# B&R Automation Studio project NAEUL004C00R13L518F00 (part 16)

#### Act_OptP0923Navi.st
```iecst
ACTION Act_OptP0923Navi:

	IF tyP0923SafetyBar.tyNaviBack.tyBtnBack.bRtCompl = TRUE OR tyP0923SafetyBar.tyNaviLyr1.tyBtnBack.bRtCompl = TRUE OR tyP0923SafetyBar.tyNaviLyr2.tyBtnBack.bRtCompl = TRUE THEN
		tyP0923SafetyBar.tyNaviBack.tyBtnBack.bRtCompl 	:= FALSE;
		tyP0923SafetyBar.tyNaviBack.tyBtnBack.bValue	:= FALSE;
		tyP0923SafetyBar.tyNaviLyr1.tyBtnBack.bRtCompl 	:= FALSE;
		tyP0923SafetyBar.tyNaviLyr1.tyBtnBack.bValue	:= FALSE;
		tyP0923SafetyBar.tyNaviLyr2.tyBtnBack.bRtCompl 	:= FALSE;
		tyP0923SafetyBar.tyNaviLyr2.tyBtnBack.bValue	:= FALSE;

		eChgPage	:= UIP0920MtrNPneuCtrl;

	ELSIF tyP0923SafetyBar.tyNaviLyr1.tyBtnLeft.bRtCompl = TRUE OR tyP0923SafetyBar.tyNaviLyr1.tyBtnRgt.bRtCompl = TRUE THEN
		tyP0923SafetyBar.tyNaviLyr1.tyBtnLeft.bRtCompl	:= FALSE;
		tyP0923SafetyBar.tyNaviLyr1.tyBtnRgt.bRtCompl	:= FALSE;

		bDispSafetyBar1	:= FALSE;
		bDispSafetyBar2	:= TRUE;

		p_tyC0004Navi ACCESS ADR(tyP0923SafetyBar.tyNaviLyr2);

		p_tyP0923LftSafetyBarCom ACCESS ADR(tyP0923SafetyBar.tyMag3SafetyBarCom);
		p_tyP0923LftSafetyBarDC ACCESS ADR(tyP0923SafetyBar.tyMag3SafetyBarDC);
		p_tyP0923LftSafetyBarFB ACCESS ADR(tyP0923SafetyBar.tyMag3SafetyBarFB);

		p_tyP0923RgtSafetyBarCom ACCESS ADR(tyP0923SafetyBar.tyRgtSafetyBarComHide);
		p_tyP0923RgtSafetyBarDC ACCESS ADR(tyP0923SafetyBar.tyRgtSafetyBarDCHide);
		p_tyP0923RgtSafetyBarFB ACCESS ADR(tyP0923SafetyBar.tyRgtSafetyBarFBHide);

	ELSIF tyP0923SafetyBar.tyNaviLyr2.tyBtnLeft.bRtCompl = TRUE OR tyP0923SafetyBar.tyNaviLyr2.tyBtnRgt.bRtCompl = TRUE THEN
		tyP0923SafetyBar.tyNaviLyr2.tyBtnLeft.bRtCompl	:= FALSE;
		tyP0923SafetyBar.tyNaviLyr2.tyBtnRgt.bRtCompl	:= FALSE;

		bDispSafetyBar1	:= TRUE;
		bDispSafetyBar2	:= FALSE;

		p_tyC0004Navi ACCESS ADR(tyP0923SafetyBar.tyNaviLyr1);

		p_tyP0923LftSafetyBarCom ACCESS ADR(tyP0923SafetyBar.tyMag1SafetyBarCom);
		p_tyP0923LftSafetyBarDC ACCESS ADR(tyP0923SafetyBar.tyMag1SafetyBarDC);
		p_tyP0923LftSafetyBarFB ACCESS ADR(tyP0923SafetyBar.tyMag1SafetyBarFB);

		p_tyP0923RgtSafetyBarCom ACCESS ADR(tyP0923SafetyBar.tyMag2SafetyBarCom);
		p_tyP0923RgtSafetyBarDC ACCESS ADR(tyP0923SafetyBar.tyMag2SafetyBarDC);
		p_tyP0923RgtSafetyBarFB ACCESS ADR(tyP0923SafetyBar.tyMag2SafetyBarFB);

	END_IF

END_ACTION
```

#### Act_OptP0923DualMask.st
```iecst
ACTION Act_OptP0923DualMask:

	IF eCurrPage = UIP0923SafetyBar THEN

		IF p_tyDI.bEStopSig = FALSE THEN
			p_tyC0003DualMask ACCESS ADR(tyP0923SafetyBar.tyDualMaskEStop);

			tyP0923SafetyBar.tyDualMaskEStop.tyBtnLeftMask.uiMaskRtStat.0	:= FALSE;
			tyP0923SafetyBar.tyDualMaskEStop.tyBtnRgtMask.uiMaskRtStat.0	:= bDispSafetyBar2;

		ELSIF p_tyDI.bCoverSWSig = FALSE THEN
			p_tyC0003DualMask ACCESS ADR(tyP0923SafetyBar.tyDualMaskCWSig);

			tyP0923SafetyBar.tyDualMaskCWSig.tyBtnLeftMask.uiMaskRtStat.0	:= FALSE;
			tyP0923SafetyBar.tyDualMaskCWSig.tyBtnRgtMask.uiMaskRtStat.0	:= bDispSafetyBar2;

		ELSIF p_tyDI.bSafetyRlySig = FALSE THEN
			p_tyC0003DualMask ACCESS ADR(tyP0923SafetyBar.tyDualMaskSafetyRly);

			tyP0923SafetyBar.tyDualMaskSafetyRly.tyBtnLeftMask.uiMaskRtStat.0	:= FALSE;
			tyP0923SafetyBar.tyDualMaskSafetyRly.tyBtnRgtMask.uiMaskRtStat.0	:= bDispSafetyBar2;

//		ELSIF p_tyDI.bPusherRetRS = FALSE THEN
//			p_tyC0003DualMask ACCESS ADR(tyP0923SafetyBar.tyDualMaskPshrInterrupt);
//
//			tyP0923SafetyBar.tyDualMaskPshrInterrupt.tyBtnLeftMask.uiMaskRtStat.0	:= FALSE;
//			tyP0923SafetyBar.tyDualMaskPshrInterrupt.tyBtnRgtMask.uiMaskRtStat.0	:= bDispSafetyBar2;
//
		ELSE
			p_tyC0003DualMask ACCESS ADR(tyP0923SafetyBar.tyDualMaskHide);

		END_IF

	END_IF

END_ACTION
```

#### Act_OptP0923Mag1SafetyBarChgLyr.st
```iecst
ACTION Act_OptP0923Mag1SafetyBarChgLyr:

	IF tyP0923SafetyBar.tyMag1SafetyBarCom.tyBtnSwitch.bRtCompl THEN
		tyP0923SafetyBar.tyMag1SafetyBarCom.tyBtnSwitch.bRtCompl := FALSE;

		IF tyP0923SafetyBar.tyMag1SafetyBarCom.tyBtnSwitch.bValue = TRUE THEN
			fUIInRtStatOff(ADR(tyP0923SafetyBar.tyMag1SafetyBarDC.tyLyr.uiRtStat));
			fUIInRtStatHide(ADR(tyP0923SafetyBar.tyMag1SafetyBarFB.tyLyr.uiRtStat));
		ELSE
			fUIInRtStatHide(ADR(tyP0923SafetyBar.tyMag1SafetyBarDC.tyLyr.uiRtStat));
			fUIInRtStatOff(ADR(tyP0923SafetyBar.tyMag1SafetyBarFB.tyLyr.uiRtStat));
		END_IF

	END_IF

END_ACTION
```

#### Act_OptP0923Mag1SafetyBarSen.st
```iecst
ACTION Act_OptP0923Mag1SafetyBarSen:

	tyP0923SafetyBar.tyMag1SafetyBarCom.tyBtnExtRS.bValue	:= p_tyDI.bMag1SafetyBarExtRS;
	tyP0923SafetyBar.tyMag1SafetyBarCom.tyBtnRetRS.bValue	:= p_tyDI.bMag1SafetyBarRetRS;

	//Machine Bitmap
	IF p_tyDI.bMag1SafetyBarRetRS = TRUE THEN
		tyP0923SafetyBar.tyMag1SafetyBarCom.tyBitmapMc.uiValueIdx	:= 1;
	ELSE
		tyP0923SafetyBar.tyMag1SafetyBarCom.tyBitmapMc.uiValueIdx	:= 0;
	END_IF

	IF p_tyNtParamCurr.eProjMag = ULMagTriple THEN
		IF p_tyNtParamCurr.bProjMagAWPrep = FALSE AND p_tyNtParamCurr.bProjMotorizedPusherPrep = FALSE THEN
		IF 	tyP0923SafetyBar.tyMag1SafetyBarCom.tyBitmapMc.uiValueIdx < 100 THEN
			tyP0923SafetyBar.tyMag1SafetyBarCom.tyBitmapMc.uiValueIdx	:= tyP0923SafetyBar.tyMag1SafetyBarCom.tyBitmapMc.uiValueIdx + 100;
		END_IF
	ELSIF p_tyNtParamCurr.bProjMagAWPrep = FALSE AND p_tyNtParamCurr.bProjMotorizedPusherPrep = TRUE THEN
		IF 	tyP0923SafetyBar.tyMag1SafetyBarCom.tyBitmapMc.uiValueIdx < 400 THEN
		tyP0923SafetyBar.tyMag1SafetyBarCom.tyBitmapMc.uiValueIdx	:= tyP0923SafetyBar.tyMag1SafetyBarCom.tyBitmapMc.uiValueIdx + 400;
		END_IF
		END_IF
		END_IF
END_ACTION
```

#### Act_OptP0923Mag1SafetyBarFB.st
```iecst
ACTION Act_OptP0923Mag1SafetyBarFB:

	IF tyP0923SafetyBar.tyMag1SafetyBarCom.tyBtnSwitch.bValue = FALSE THEN

		IF tyP0923SafetyBar.tyMag1SafetyBarFB.tyBtnRet.bRtCompl = TRUE THEN
			tyP0923SafetyBar.tyMag1SafetyBarFB.tyBtnRet.bRtCompl	:= FALSE;

			tyP0923SafetyBar.tyMag1SafetyBarFB.tyBtnRet.bValue		:= TRUE;
			tyP0923SafetyBar.tyMag1SafetyBarFB.tyBtnExt.bValue		:= FALSE;

		ELSIF tyP0923SafetyBar.tyMag1SafetyBarFB.tyBtnExt.bRtCompl = TRUE THEN
			tyP0923SafetyBar.tyMag1SafetyBarFB.tyBtnExt.bRtCompl	:= FALSE;

			tyP0923SafetyBar.tyMag1SafetyBarFB.tyBtnExt.bValue		:= TRUE;
			tyP0923SafetyBar.tyMag1SafetyBarFB.tyBtnRet.bValue		:= FALSE;
		END_IF

		IF tyP0923SafetyBar.tyMag1SafetyBarFB.tyBtnRet.bValue = TRUE THEN
			eMag1SafetyBarAct	:= PneuActRet;

			IF p_eMag1SafetyBarStat = PneuActRet AND p_eMag1SafetyBarStatus = Done THEN
				eMag1SafetyBarAct	:= PneuActIdle;

				tyP0923SafetyBar.tyMag1SafetyBarFB.tyBtnRet.bValue	:= FALSE;
			ELSIF p_eMag1SafetyBarStatus = Error THEN
				tyP0923SafetyBar.tyMag1SafetyBarFB.tyBtnRet.bValue	:= FALSE;
			END_IF

		ELSIF tyP0923SafetyBar.tyMag1SafetyBarFB.tyBtnExt.bValue = TRUE THEN
			eMag1SafetyBarAct	:= PneuActExt;

			IF p_eMag1SafetyBarStat = PneuActExt AND p_eMag1SafetyBarStatus = Done THEN
				eMag1SafetyBarAct	:= PneuActIdle;

				tyP0923SafetyBar.tyMag1SafetyBarFB.tyBtnExt.bValue := FALSE;
			ELSIF p_eMag1SafetyBarStatus = Error THEN
				tyP0923SafetyBar.tyMag1SafetyBarFB.tyBtnExt.bValue := FALSE;
			END_IF
		END_IF

		//Update Direct Control Status
		tyP0923SafetyBar.tyMag1SafetyBarDC.tyBtnRet.bRtCompl	:= FALSE;
		tyP0923SafetyBar.tyMag1SafetyBarDC.tyBtnExt.bRtCompl	:= FALSE;
		tyP0923SafetyBar.tyMag1SafetyBarDC.tyBtnRet.bValue		:= p_bMag1SafetyBarRetCtrl;
		tyP0923SafetyBar.tyMag1SafetyBarDC.tyBtnExt.bValue		:= p_bMag1SafetyBarExtCtrl;

	END_IF

END_ACTION
```

#### Act_OptP0923Mag1SafetyBarFBStat.st
```iecst
ACTION Act_OptP0923Mag1SafetyBarFBStat:

	tyP0923SafetyBar.tyMag1SafetyBarFB.tyStringStat.sValue	:= p_sMag1SafetyBarStatTxt;

END_ACTION
```

#### Act_OptP0923Mag1SafetyBarDC.st
```iecst
ACTION Act_OptP0923Mag1SafetyBarDC:

	IF tyP0923SafetyBar.tyMag1SafetyBarCom.tyBtnSwitch.bValue = TRUE THEN

		IF p_bMag1SafetyBarTwoCtrlOut = FALSE THEN

			IF tyP0923SafetyBar.tyMag1SafetyBarDC.tyBtnRet.bRtCompl = TRUE THEN
				tyP0923SafetyBar.tyMag1SafetyBarDC.tyBtnRet.bValue	:= TRUE;
				tyP0923SafetyBar.tyMag1SafetyBarDC.tyBtnExt.bValue	:= FALSE;

				eMag1SafetyBarAct	:= PneuActSetRet;

				IF p_eMag1SafetyBarStat = PneuActSetRet AND p_eMag1SafetyBarStatus = Done THEN
					eMag1SafetyBarAct	:= PneuActIdle;

					tyP0923SafetyBar.tyMag1SafetyBarDC.tyBtnRet.bRtCompl	:= FALSE;
				END_IF

			ELSIF tyP0923SafetyBar.tyMag1SafetyBarDC.tyBtnExt.bRtCompl = TRUE THEN
				tyP0923SafetyBar.tyMag1SafetyBarDC.tyBtnExt.bValue	:= TRUE;
				tyP0923SafetyBar.tyMag1SafetyBarDC.tyBtnRet.bValue	:= FALSE;

				eMag1SafetyBarAct	:= PneuActSetExt;

				IF p_eMag1SafetyBarStat = PneuActSetExt AND p_eMag1SafetyBarStatus = Done THEN
					eMag1SafetyBarAct	:= PneuActIdle;

					tyP0923SafetyBar.tyMag1SafetyBarDC.tyBtnExt.bRtCompl	:= FALSE;
				END_IF

			END_IF

		ELSE

			IF (tyP0923SafetyBar.tyMag1SafetyBarDC.tyBtnRet.bRtCompl = TRUE) OR (tyP0923SafetyBar.tyMag1SafetyBarDC.tyBtnExt.bRtCompl = TRUE) THEN

				IF (tyP0923SafetyBar.tyMag1SafetyBarDC.tyBtnRet.bValue = TRUE) AND (tyP0923SafetyBar.tyMag1SafetyBarDC.tyBtnExt.bValue = TRUE) THEN
					eMag1SafetyBarAct	:= PneuActSetAll;

					IF p_eMag1SafetyBarStat = PneuActSetAll AND p_eMag1SafetyBarStatus = Done THEN
						eMag1SafetyBarAct	:= PneuActIdle;

						tyP0923SafetyBar.tyMag1SafetyBarDC.tyBtnRet.bRtCompl	:= FALSE;
						tyP0923SafetyBar.tyMag1SafetyBarDC.tyBtnExt.bRtCompl	:= FALSE;
					END_IF

				ELSIF (tyP0923SafetyBar.tyMag1SafetyBarDC.tyBtnRet.bValue = TRUE) AND (tyP0923SafetyBar.tyMag1SafetyBarDC.tyBtnExt.bValue = FALSE) THEN
					eMag1SafetyBarAct	:= PneuActSetRet;

					IF p_eMag1SafetyBarStat = PneuActSetRet AND p_eMag1SafetyBarStatus = Done THEN
						eMag1SafetyBarAct	:= PneuActIdle;

						tyP0923SafetyBar.tyMag1SafetyBarDC.tyBtnRet.bRtCompl	:= FALSE;
						tyP0923SafetyBar.tyMag1SafetyBarDC.tyBtnExt.bRtCompl	:= FALSE;
					END_IF

				ELSIF (tyP0923SafetyBar.tyMag1SafetyBarDC.tyBtnRet.bValue = FALSE) AND (tyP0923SafetyBar.tyMag1SafetyBarDC.tyBtnExt.bValue = TRUE) THEN
					eMag1SafetyBarAct	:= PneuActSetExt;

					IF p_eMag1SafetyBarStat = PneuActSetExt AND p_eMag1SafetyBarStatus = Done THEN
						eMag1SafetyBarAct	:= PneuActIdle;

						tyP0923SafetyBar.tyMag1SafetyBarDC.tyBtnRet.bRtCompl	:= FALSE;
						tyP0923SafetyBar.tyMag1SafetyBarDC.tyBtnExt.bRtCompl	:= FALSE;
					END_IF

				ELSE
					eMag1SafetyBarAct	:= PneuActRstAll;

					IF p_eMag1SafetyBarStat = PneuActRstAll AND p_eMag1SafetyBarStatus = Done THEN
						eMag1SafetyBarAct	:= PneuActIdle;

						tyP0923SafetyBar.tyMag1SafetyBarDC.tyBtnRet.bRtCompl	:= FALSE;
						tyP0923SafetyBar.tyMag1SafetyBarDC.tyBtnExt.bRtCompl	:= FALSE;
					END_IF

				END_IF

			END_IF

		END_IF

		tyP0923SafetyBar.tyMag1SafetyBarFB.tyBtnExt.bRtCompl	:= FALSE;
		tyP0923SafetyBar.tyMag1SafetyBarFB.tyBtnExt.bValue		:= FALSE;
		tyP0923SafetyBar.tyMag1SafetyBarFB.tyBtnRet.bRtCompl	:= FALSE;
		tyP0923SafetyBar.tyMag1SafetyBarFB.tyBtnRet.bValue		:= FALSE;

	END_IF

END_ACTION
```

#### Act_OptP0923Mag2SafetyBarChgLyr.st
```iecst
ACTION Act_OptP0923Mag2SafetyBarChgLyr:

	IF tyP0923SafetyBar.tyMag2SafetyBarCom.tyBtnSwitch.bRtCompl THEN
		tyP0923SafetyBar.tyMag2SafetyBarCom.tyBtnSwitch.bRtCompl := FALSE;

		IF tyP0923SafetyBar.tyMag2SafetyBarCom.tyBtnSwitch.bValue = TRUE THEN
			fUIInRtStatOff(ADR(tyP0923SafetyBar.tyMag2SafetyBarDC.tyLyr.uiRtStat));
			fUIInRtStatHide(ADR(tyP0923SafetyBar.tyMag2SafetyBarFB.tyLyr.uiRtStat));
		ELSE
			fUIInRtStatHide(ADR(tyP0923SafetyBar.tyMag2SafetyBarDC.tyLyr.uiRtStat));
			fUIInRtStatOff(ADR(tyP0923SafetyBar.tyMag2SafetyBarFB.tyLyr.uiRtStat));
		END_IF

	END_IF

END_ACTION
```

#### Act_OptP0923Mag2SafetyBarSen.st
```iecst
ACTION Act_OptP0923Mag2SafetyBarSen:

	tyP0923SafetyBar.tyMag2SafetyBarCom.tyBtnExtRS.bValue	:= p_tyDI.bMag2SafetyBarExtRS;
	tyP0923SafetyBar.tyMag2SafetyBarCom.tyBtnRetRS.bValue	:= p_tyDI.bMag2SafetyBarRetRS;

	//Machine Bitmap
	IF p_tyDI.bMag2SafetyBarRetRS = TRUE THEN
		tyP0923SafetyBar.tyMag2SafetyBarCom.tyBitmapMc.uiValueIdx	:= 3;
	ELSE
		tyP0923SafetyBar.tyMag2SafetyBarCom.tyBitmapMc.uiValueIdx	:= 2;
	END_IF

	IF p_tyNtParamCurr.eProjMag = ULMagTriple THEN
		IF p_tyNtParamCurr.bProjMagAWPrep = FALSE AND p_tyNtParamCurr.bProjMotorizedPusherPrep = FALSE THEN
		IF 	tyP0923SafetyBar.tyMag2SafetyBarCom.tyBitmapMc.uiValueIdx < 100 THEN
				tyP0923SafetyBar.tyMag2SafetyBarCom.tyBitmapMc.usiValueIdx	:= tyP0923SafetyBar.tyMag2SafetyBarCom.tyBitmapMc.usiValueIdx + 100;
				END_IF
	ELSIF p_tyNtParamCurr.bProjMagAWPrep = FALSE AND p_tyNtParamCurr.bProjMotorizedPusherPrep = TRUE THEN
		IF 	tyP0923SafetyBar.tyMag2SafetyBarCom.tyBitmapMc.uiValueIdx < 400 THEN
			tyP0923SafetyBar.tyMag2SafetyBarCom.tyBitmapMc.uiValueIdx	:= tyP0923SafetyBar.tyMag2SafetyBarCom.tyBitmapMc.uiValueIdx + 400;
		END_IF
			END_IF
			END_IF
END_ACTION
```

#### Act_OptP0923Mag2SafetyBarFB.st
```iecst
ACTION Act_OptP0923Mag2SafetyBarFB:

	IF tyP0923SafetyBar.tyMag2SafetyBarCom.tyBtnSwitch.bValue = FALSE THEN

		IF tyP0923SafetyBar.tyMag2SafetyBarFB.tyBtnRet.bRtCompl = TRUE THEN
			tyP0923SafetyBar.tyMag2SafetyBarFB.tyBtnRet.bRtCompl	:= FALSE;

			tyP0923SafetyBar.tyMag2SafetyBarFB.tyBtnRet.bValue		:= TRUE;
			tyP0923SafetyBar.tyMag2SafetyBarFB.tyBtnExt.bValue		:= FALSE;

		ELSIF tyP0923SafetyBar.tyMag2SafetyBarFB.tyBtnExt.bRtCompl = TRUE THEN
			tyP0923SafetyBar.tyMag2SafetyBarFB.tyBtnExt.bRtCompl	:= FALSE;

			tyP0923SafetyBar.tyMag2SafetyBarFB.tyBtnExt.bValue		:= TRUE;
			tyP0923SafetyBar.tyMag2SafetyBarFB.tyBtnRet.bValue		:= FALSE;
		END_IF

		IF tyP0923SafetyBar.tyMag2SafetyBarFB.tyBtnRet.bValue = TRUE THEN
			eMag2SafetyBarAct	:= PneuActRet;

			IF p_eMag2SafetyBarStat = PneuActRet AND p_eMag2SafetyBarStatus = Done THEN
				eMag2SafetyBarAct	:= PneuActIdle;

				tyP0923SafetyBar.tyMag2SafetyBarFB.tyBtnRet.bValue	:= FALSE;
			ELSIF p_eMag2SafetyBarStatus = Error THEN
				tyP0923SafetyBar.tyMag2SafetyBarFB.tyBtnRet.bValue	:= FALSE;
			END_IF

		ELSIF tyP0923SafetyBar.tyMag2SafetyBarFB.tyBtnExt.bValue = TRUE THEN
			eMag2SafetyBarAct	:= PneuActExt;

			IF p_eMag2SafetyBarStat = PneuActExt AND p_eMag2SafetyBarStatus = Done THEN
				eMag2SafetyBarAct	:= PneuActIdle;

				tyP0923SafetyBar.tyMag2SafetyBarFB.tyBtnExt.bValue := FALSE;
			ELSIF p_eMag2SafetyBarStatus = Error THEN
				tyP0923SafetyBar.tyMag2SafetyBarFB.tyBtnExt.bValue := FALSE;
			END_IF
		END_IF

		//Update Direct Control Status
		tyP0923SafetyBar.tyMag2SafetyBarDC.tyBtnRet.bRtCompl	:= FALSE;
		tyP0923SafetyBar.tyMag2SafetyBarDC.tyBtnExt.bRtCompl	:= FALSE;
		tyP0923SafetyBar.tyMag2SafetyBarDC.tyBtnRet.bValue		:= p_bMag2SafetyBarRetCtrl;
		tyP0923SafetyBar.tyMag2SafetyBarDC.tyBtnExt.bValue		:= p_bMag2SafetyBarExtCtrl;

	END_IF

END_ACTION
```

#### Act_OptP0923Mag2SafetyBarFBStat.st
```iecst
ACTION Act_OptP0923Mag2SafetyBarFBStat:

	tyP0923SafetyBar.tyMag2SafetyBarFB.tyStringStat.sValue	:= p_sMag2SafetyBarStatTxt;

END_ACTION
```

#### Act_OptP0923Mag2SafetyBarDC.st
```iecst
ACTION Act_OptP0923Mag2SafetyBarDC:

	IF tyP0923SafetyBar.tyMag2SafetyBarCom.tyBtnSwitch.bValue = TRUE THEN

		IF p_bMag2SafetyBarTwoCtrlOut = FALSE THEN

			IF tyP0923SafetyBar.tyMag2SafetyBarDC.tyBtnRet.bRtCompl = TRUE THEN
				tyP0923SafetyBar.tyMag2SafetyBarDC.tyBtnRet.bValue	:= TRUE;
				tyP0923SafetyBar.tyMag2SafetyBarDC.tyBtnExt.bValue	:= FALSE;

				eMag2SafetyBarAct	:= PneuActSetRet;

				IF p_eMag2SafetyBarStat = PneuActSetRet AND p_eMag2SafetyBarStatus = Done THEN
					eMag2SafetyBarAct	:= PneuActIdle;

					tyP0923SafetyBar.tyMag2SafetyBarDC.tyBtnRet.bRtCompl	:= FALSE;
				END_IF

			ELSIF tyP0923SafetyBar.tyMag2SafetyBarDC.tyBtnExt.bRtCompl = TRUE THEN
				tyP0923SafetyBar.tyMag2SafetyBarDC.tyBtnExt.bValue	:= TRUE;
				tyP0923SafetyBar.tyMag2SafetyBarDC.tyBtnRet.bValue	:= FALSE;

				eMag2SafetyBarAct	:= PneuActSetExt;

				IF p_eMag2SafetyBarStat = PneuActSetExt AND p_eMag2SafetyBarStatus = Done THEN
					eMag2SafetyBarAct	:= PneuActIdle;

					tyP0923SafetyBar.tyMag2SafetyBarDC.tyBtnExt.bRtCompl	:= FALSE;
				END_IF

			END_IF

		ELSE

			IF (tyP0923SafetyBar.tyMag2SafetyBarDC.tyBtnRet.bRtCompl = TRUE) OR (tyP0923SafetyBar.tyMag2SafetyBarDC.tyBtnExt.bRtCompl = TRUE) THEN

				IF (tyP0923SafetyBar.tyMag2SafetyBarDC.tyBtnRet.bValue = TRUE) AND (tyP0923SafetyBar.tyMag2SafetyBarDC.tyBtnExt.bValue = TRUE) THEN
					eMag2SafetyBarAct	:= PneuActSetAll;

					IF p_eMag2SafetyBarStat = PneuActSetAll AND p_eMag2SafetyBarStatus = Done THEN
						eMag2SafetyBarAct	:= PneuActIdle;

						tyP0923SafetyBar.tyMag2SafetyBarDC.tyBtnRet.bRtCompl	:= FALSE;
						tyP0923SafetyBar.tyMag2SafetyBarDC.tyBtnExt.bRtCompl	:= FALSE;
					END_IF

				ELSIF (tyP0923SafetyBar.tyMag2SafetyBarDC.tyBtnRet.bValue = TRUE) AND (tyP0923SafetyBar.tyMag2SafetyBarDC.tyBtnExt.bValue = FALSE) THEN
					eMag2SafetyBarAct	:= PneuActSetRet;

					IF p_eMag2SafetyBarStat = PneuActSetRet AND p_eMag2SafetyBarStatus = Done THEN
						eMag2SafetyBarAct	:= PneuActIdle;

						tyP0923SafetyBar.tyMag2SafetyBarDC.tyBtnRet.bRtCompl	:= FALSE;
						tyP0923SafetyBar.tyMag2SafetyBarDC.tyBtnExt.bRtCompl	:= FALSE;
					END_IF

				ELSIF (tyP0923SafetyBar.tyMag2SafetyBarDC.tyBtnRet.bValue = FALSE) AND (tyP0923SafetyBar.tyMag2SafetyBarDC.tyBtnExt.bValue = TRUE) THEN
					eMag2SafetyBarAct	:= PneuActSetExt;

					IF p_eMag2SafetyBarStat = PneuActSetExt AND p_eMag2SafetyBarStatus = Done THEN
						eMag2SafetyBarAct	:= PneuActIdle;

						tyP0923SafetyBar.tyMag2SafetyBarDC.tyBtnRet.bRtCompl	:= FALSE;
						tyP0923SafetyBar.tyMag2SafetyBarDC.tyBtnExt.bRtCompl	:= FALSE;
					END_IF

				ELSE
					eMag2SafetyBarAct	:= PneuActRstAll;

					IF p_eMag2SafetyBarStat = PneuActRstAll AND p_eMag2SafetyBarStatus = Done THEN
						eMag2SafetyBarAct	:= PneuActIdle;

						tyP0923SafetyBar.tyMag2SafetyBarDC.tyBtnRet.bRtCompl	:= FALSE;
						tyP0923SafetyBar.tyMag2SafetyBarDC.tyBtnExt.bRtCompl	:= FALSE;
					END_IF

				END_IF

			END_IF

		END_IF

		tyP0923SafetyBar.tyMag2SafetyBarFB.tyBtnExt.bRtCompl	:= FALSE;
		tyP0923SafetyBar.tyMag2SafetyBarFB.tyBtnExt.bValue		:= FALSE;
		tyP0923SafetyBar.tyMag2SafetyBarFB.tyBtnRet.bRtCompl	:= FALSE;
		tyP0923SafetyBar.tyMag2SafetyBarFB.tyBtnRet.bValue		:= FALSE;

	END_IF

END_ACTION
```

#### Act_OptP0923Mag3SafetyBarChgLyr.st
```iecst
ACTION Act_OptP0923Mag3SafetyBarChgLyr:

	IF tyP0923SafetyBar.tyMag3SafetyBarCom.tyBtnSwitch.bRtCompl THEN
		tyP0923SafetyBar.tyMag3SafetyBarCom.tyBtnSwitch.bRtCompl := FALSE;

		IF tyP0923SafetyBar.tyMag3SafetyBarCom.tyBtnSwitch.bValue = TRUE THEN
			fUIInRtStatOff(ADR(tyP0923SafetyBar.tyMag3SafetyBarDC.tyLyr.uiRtStat));
			fUIInRtStatHide(ADR(tyP0923SafetyBar.tyMag3SafetyBarFB.tyLyr.uiRtStat));
		ELSE
			fUIInRtStatHide(ADR(tyP0923SafetyBar.tyMag3SafetyBarDC.tyLyr.uiRtStat));
			fUIInRtStatOff(ADR(tyP0923SafetyBar.tyMag3SafetyBarFB.tyLyr.uiRtStat));
		END_IF

	END_IF

END_ACTION
```

#### Act_OptP0923Mag3SafetyBarSen.st
```iecst
ACTION Act_OptP0923Mag3SafetyBarSen:

	tyP0923SafetyBar.tyMag3SafetyBarCom.tyBtnExtRS.bValue	:= p_tyDI.bMag3SafetyBarExtRS;
	tyP0923SafetyBar.tyMag3SafetyBarCom.tyBtnRetRS.bValue	:= p_tyDI.bMag3SafetyBarRetRS;

	//Machine Bitmap
	IF p_tyDI.bMag3SafetyBarRetRS = TRUE THEN
		tyP0923SafetyBar.tyMag3SafetyBarCom.tyBitmapMc.uiValueIdx	:= 5;
	ELSE
		tyP0923SafetyBar.tyMag3SafetyBarCom.tyBitmapMc.uiValueIdx	:= 4;
	END_IF

	IF p_tyNtParamCurr.eProjMag = ULMagTriple THEN
		IF p_tyNtParamCurr.bProjMagAWPrep = FALSE AND p_tyNtParamCurr.bProjMotorizedPusherPrep = FALSE THEN
		IF 	tyP0923SafetyBar.tyMag3SafetyBarCom.tyBitmapMc.uiValueIdx < 100 THEN
		tyP0923SafetyBar.tyMag3SafetyBarCom.tyBitmapMc.usiValueIdx	:= tyP0923SafetyBar.tyMag3SafetyBarCom.tyBitmapMc.usiValueIdx + 100;
		END_IF
		ELSIF p_tyNtParamCurr.bProjMagAWPrep = FALSE AND p_tyNtParamCurr.bProjMotorizedPusherPrep = TRUE THEN
		IF 	tyP0923SafetyBar.tyMag3SafetyBarCom.tyBitmapMc.uiValueIdx < 400 THEN
			tyP0923SafetyBar.tyMag3SafetyBarCom.tyBitmapMc.uiValueIdx	:= tyP0923SafetyBar.tyMag3SafetyBarCom.tyBitmapMc.uiValueIdx + 400;
		END_IF
		END_IF
		END_IF
END_ACTION
```

#### Act_OptP0923Mag3SafetyBarFB.st
```iecst
ACTION Act_OptP0923Mag3SafetyBarFB:

	IF tyP0923SafetyBar.tyMag3SafetyBarCom.tyBtnSwitch.bValue = FALSE THEN

		IF tyP0923SafetyBar.tyMag3SafetyBarFB.tyBtnRet.bRtCompl = TRUE THEN
			tyP0923SafetyBar.tyMag3SafetyBarFB.tyBtnRet.bRtCompl	:= FALSE;

			tyP0923SafetyBar.tyMag3SafetyBarFB.tyBtnRet.bValue		:= TRUE;
			tyP0923SafetyBar.tyMag3SafetyBarFB.tyBtnExt.bValue		:= FALSE;

		ELSIF tyP0923SafetyBar.tyMag3SafetyBarFB.tyBtnExt.bRtCompl = TRUE THEN
			tyP0923SafetyBar.tyMag3SafetyBarFB.tyBtnExt.bRtCompl	:= FALSE;

			tyP0923SafetyBar.tyMag3SafetyBarFB.tyBtnExt.bValue		:= TRUE;
			tyP0923SafetyBar.tyMag3SafetyBarFB.tyBtnRet.bValue		:= FALSE;
		END_IF

		IF tyP0923SafetyBar.tyMag3SafetyBarFB.tyBtnRet.bValue = TRUE THEN
			eMag3SafetyBarAct	:= PneuActRet;

			IF p_eMag3SafetyBarStat = PneuActRet AND p_eMag3SafetyBarStatus = Done THEN
				eMag3SafetyBarAct	:= PneuActIdle;

				tyP0923SafetyBar.tyMag3SafetyBarFB.tyBtnRet.bValue	:= FALSE;
			ELSIF p_eMag3SafetyBarStatus = Error THEN
				tyP0923SafetyBar.tyMag3SafetyBarFB.tyBtnRet.bValue	:= FALSE;
			END_IF

		ELSIF tyP0923SafetyBar.tyMag3SafetyBarFB.tyBtnExt.bValue = TRUE THEN
			eMag3SafetyBarAct	:= PneuActExt;

			IF p_eMag3SafetyBarStat = PneuActExt AND p_eMag3SafetyBarStatus = Done THEN
				eMag3SafetyBarAct	:= PneuActIdle;

				tyP0923SafetyBar.tyMag3SafetyBarFB.tyBtnExt.bValue := FALSE;
			ELSIF p_eMag3SafetyBarStatus = Error THEN
				tyP0923SafetyBar.tyMag3SafetyBarFB.tyBtnExt.bValue := FALSE;
			END_IF
		END_IF

		//Update Direct Control Status
		tyP0923SafetyBar.tyMag3SafetyBarDC.tyBtnRet.bRtCompl	:= FALSE;
		tyP0923SafetyBar.tyMag3SafetyBarDC.tyBtnExt.bRtCompl	:= FALSE;
		tyP0923SafetyBar.tyMag3SafetyBarDC.tyBtnRet.bValue		:= p_bMag3SafetyBarRetCtrl;
		tyP0923SafetyBar.tyMag3SafetyBarDC.tyBtnExt.bValue		:= p_bMag3SafetyBarExtCtrl;

	END_IF

END_ACTION
```

#### Act_OptP0923Mag3SafetyBarFBStat.st
```iecst
ACTION Act_OptP0923Mag3SafetyBarFBStat:

	tyP0923SafetyBar.tyMag3SafetyBarFB.tyStringStat.sValue	:= p_sMag3SafetyBarStatTxt;

END_ACTION
```

#### Act_OptP0923Mag3SafetyBarDC.st
```iecst
ACTION Act_OptP0923Mag3SafetyBarDC:

	IF tyP0923SafetyBar.tyMag3SafetyBarCom.tyBtnSwitch.bValue = TRUE THEN

		IF p_bMag3SafetyBarTwoCtrlOut = FALSE THEN

			IF tyP0923SafetyBar.tyMag3SafetyBarDC.tyBtnRet.bRtCompl = TRUE THEN
				tyP0923SafetyBar.tyMag3SafetyBarDC.tyBtnRet.bValue	:= TRUE;
				tyP0923SafetyBar.tyMag3SafetyBarDC.tyBtnExt.bValue	:= FALSE;

				eMag3SafetyBarAct	:= PneuActSetRet;

				IF p_eMag3SafetyBarStat = PneuActSetRet AND p_eMag3SafetyBarStatus = Done THEN
					eMag3SafetyBarAct	:= PneuActIdle;

					tyP0923SafetyBar.tyMag3SafetyBarDC.tyBtnRet.bRtCompl	:= FALSE;
				END_IF

			ELSIF tyP0923SafetyBar.tyMag3SafetyBarDC.tyBtnExt.bRtCompl = TRUE THEN
				tyP0923SafetyBar.tyMag3SafetyBarDC.tyBtnExt.bValue	:= TRUE;
				tyP0923SafetyBar.tyMag3SafetyBarDC.tyBtnRet.bValue	:= FALSE;

				eMag3SafetyBarAct	:= PneuActSetExt;

				IF p_eMag3SafetyBarStat = PneuActSetExt AND p_eMag3SafetyBarStatus = Done THEN
					eMag3SafetyBarAct	:= PneuActIdle;

					tyP0923SafetyBar.tyMag3SafetyBarDC.tyBtnExt.bRtCompl	:= FALSE;
				END_IF

			END_IF

		ELSE

			IF (tyP0923SafetyBar.tyMag3SafetyBarDC.tyBtnRet.bRtCompl = TRUE) OR (tyP0923SafetyBar.tyMag3SafetyBarDC.tyBtnExt.bRtCompl = TRUE) THEN

				IF (tyP0923SafetyBar.tyMag3SafetyBarDC.tyBtnRet.bValue = TRUE) AND (tyP0923SafetyBar.tyMag3SafetyBarDC.tyBtnExt.bValue = TRUE) THEN
					eMag3SafetyBarAct	:= PneuActSetAll;

					IF p_eMag3SafetyBarStat = PneuActSetAll AND p_eMag3SafetyBarStatus = Done THEN
						eMag3SafetyBarAct	:= PneuActIdle;

						tyP0923SafetyBar.tyMag3SafetyBarDC.tyBtnRet.bRtCompl	:= FALSE;
						tyP0923SafetyBar.tyMag3SafetyBarDC.tyBtnExt.bRtCompl	:= FALSE;
					END_IF

				ELSIF (tyP0923SafetyBar.tyMag3SafetyBarDC.tyBtnRet.bValue = TRUE) AND (tyP0923SafetyBar.tyMag3SafetyBarDC.tyBtnExt.bValue = FALSE) THEN
					eMag3SafetyBarAct	:= PneuActSetRet;

					IF p_eMag3SafetyBarStat = PneuActSetRet AND p_eMag3SafetyBarStatus = Done THEN
						eMag3SafetyBarAct	:= PneuActIdle;

						tyP0923SafetyBar.tyMag3SafetyBarDC.tyBtnRet.bRtCompl	:= FALSE;
						tyP0923SafetyBar.tyMag3SafetyBarDC.tyBtnExt.bRtCompl	:= FALSE;
					END_IF

				ELSIF (tyP0923SafetyBar.tyMag3SafetyBarDC.tyBtnRet.bValue = FALSE) AND (tyP0923SafetyBar.tyMag3SafetyBarDC.tyBtnExt.bValue = TRUE) THEN
					eMag3SafetyBarAct	:= PneuActSetExt;

					IF p_eMag3SafetyBarStat = PneuActSetExt AND p_eMag3SafetyBarStatus = Done THEN
						eMag3SafetyBarAct	:= PneuActIdle;

						tyP0923SafetyBar.tyMag3SafetyBarDC.tyBtnRet.bRtCompl	:= FALSE;
						tyP0923SafetyBar.tyMag3SafetyBarDC.tyBtnExt.bRtCompl	:= FALSE;
					END_IF

				ELSE
					eMag3SafetyBarAct	:= PneuActRstAll;

					IF p_eMag3SafetyBarStat = PneuActRstAll AND p_eMag3SafetyBarStatus = Done THEN
						eMag3SafetyBarAct	:= PneuActIdle;

						tyP0923SafetyBar.tyMag3SafetyBarDC.tyBtnRet.bRtCompl	:= FALSE;
						tyP0923SafetyBar.tyMag3SafetyBarDC.tyBtnExt.bRtCompl	:= FALSE;
					END_IF

				END_IF

			END_IF

		END_IF

		tyP0923SafetyBar.tyMag3SafetyBarFB.tyBtnExt.bRtCompl	:= FALSE;
		tyP0923SafetyBar.tyMag3SafetyBarFB.tyBtnExt.bValue		:= FALSE;
		tyP0923SafetyBar.tyMag3SafetyBarFB.tyBtnRet.bRtCompl	:= FALSE;
		tyP0923SafetyBar.tyMag3SafetyBarFB.tyBtnRet.bValue		:= FALSE;

	END_IF

END_ACTION
```

#### Act_OptP0923RstMnl.st
```iecst
ACTION Act_OptP0923RstMnl:

	IF EDGEPOS((bManualMod = FALSE) OR (p_eMag1SafetyBarStatus = Error)) THEN

		eMag1SafetyBarAct	:= PneuActIdle;

		tyP0923SafetyBar.tyMag1SafetyBarDC.tyBtnRet.bRtCompl	:= FALSE;
		tyP0923SafetyBar.tyMag1SafetyBarDC.tyBtnRet.bValue		:= FALSE;
		tyP0923SafetyBar.tyMag1SafetyBarDC.tyBtnExt.bRtCompl	:= FALSE;
		tyP0923SafetyBar.tyMag1SafetyBarDC.tyBtnExt.bValue		:= FALSE;

		tyP0923SafetyBar.tyMag1SafetyBarFB.tyBtnRet.bRtCompl	:= FALSE;
		tyP0923SafetyBar.tyMag1SafetyBarFB.tyBtnRet.bValue		:= FALSE;
		tyP0923SafetyBar.tyMag1SafetyBarFB.tyBtnExt.bRtCompl	:= FALSE;
		tyP0923SafetyBar.tyMag1SafetyBarFB.tyBtnExt.bValue		:= FALSE;

	END_IF

	IF EDGEPOS((bManualMod = FALSE) OR (p_eMag2SafetyBarStatus = Error)) THEN

		eMag2SafetyBarAct	:= PneuActIdle;

		tyP0923SafetyBar.tyMag2SafetyBarDC.tyBtnRet.bRtCompl	:= FALSE;
		tyP0923SafetyBar.tyMag2SafetyBarDC.tyBtnRet.bValue		:= FALSE;
		tyP0923SafetyBar.tyMag2SafetyBarDC.tyBtnExt.bRtCompl	:= FALSE;
		tyP0923SafetyBar.tyMag2SafetyBarDC.tyBtnExt.bValue		:= FALSE;

		tyP0923SafetyBar.tyMag2SafetyBarFB.tyBtnRet.bRtCompl	:= FALSE;
		tyP0923SafetyBar.tyMag2SafetyBarFB.tyBtnRet.bValue		:= FALSE;
		tyP0923SafetyBar.tyMag2SafetyBarFB.tyBtnExt.bRtCompl	:= FALSE;
		tyP0923SafetyBar.tyMag2SafetyBarFB.tyBtnExt.bValue		:= FALSE;

	END_IF

	IF EDGEPOS((bManualMod = FALSE) OR (p_eMag3SafetyBarStatus = Error)) THEN

		eMag3SafetyBarAct	:= PneuActIdle;

		tyP0923SafetyBar.tyMag3SafetyBarDC.tyBtnRet.bRtCompl	:= FALSE;
		tyP0923SafetyBar.tyMag3SafetyBarDC.tyBtnRet.bValue		:= FALSE;
		tyP0923SafetyBar.tyMag3SafetyBarDC.tyBtnExt.bRtCompl	:= FALSE;
		tyP0923SafetyBar.tyMag3SafetyBarDC.tyBtnExt.bValue		:= FALSE;

		tyP0923SafetyBar.tyMag3SafetyBarFB.tyBtnRet.bRtCompl	:= FALSE;
		tyP0923SafetyBar.tyMag3SafetyBarFB.tyBtnRet.bValue		:= FALSE;
		tyP0923SafetyBar.tyMag3SafetyBarFB.tyBtnExt.bRtCompl	:= FALSE;
		tyP0923SafetyBar.tyMag3SafetyBarFB.tyBtnExt.bValue		:= FALSE;

	END_IF

	IF EDGEPOS(bManualMod = FALSE) THEN
		tyP0923SafetyBar.tyMag1SafetyBarCom.tyBtnSwitch.bValue := FALSE;
		tyP0923SafetyBar.tyMag2SafetyBarCom.tyBtnSwitch.bValue := FALSE;
		tyP0923SafetyBar.tyMag3SafetyBarCom.tyBtnSwitch.bValue := FALSE;

		fUIInRtStatHide(ADR(tyP0923SafetyBar.tyMag1SafetyBarDC.tyLyr.uiRtStat));
		fUIInRtStatOff(ADR(tyP0923SafetyBar.tyMag1SafetyBarFB.tyLyr.uiRtStat));

		fUIInRtStatHide(ADR(tyP0923SafetyBar.tyMag2SafetyBarDC.tyLyr.uiRtStat));
		fUIInRtStatOff(ADR(tyP0923SafetyBar.tyMag2SafetyBarFB.tyLyr.uiRtStat));

		fUIInRtStatHide(ADR(tyP0923SafetyBar.tyMag3SafetyBarDC.tyLyr.uiRtStat));
		fUIInRtStatOff(ADR(tyP0923SafetyBar.tyMag3SafetyBarFB.tyLyr.uiRtStat));
	END_IF

END_ACTION
```

#### Act_EntP0926Disp.st
```iecst
ACTION Act_EntP0926Disp:

	// Access Address
	p_tyC0002FullMask ACCESS ADR(tyP0926LifterMagConv.tyFullMaskHide);

	p_tyC0004Navi ACCESS ADR(tyP0926LifterMagConv.tyNaviBack);

	p_tyC0005Main ACCESS ADR(tyCommon.tyMain);

	p_tyC0007Notif ACCESS ADR(tyCommon.tyNotif);

	p_tyC0008MsgBox ACCESS ADR(tyP0926LifterMagConv.tyMsgBoxHide);

	p_tyC0009Info ACCESS ADR(tyCommon.tyInfo);

	p_tyP0926LifterMagConvCom ACCESS ADR(tyP0926LifterMagConv.tyCom);
	p_tyP0926LifterMagConvDC ACCESS ADR(tyP0926LifterMagConv.tyDC);
	p_tyP0926LifterMagConvFB ACCESS ADR(tyP0926LifterMagConv.tyFB);

	// Display
//	IF p_tyDI.bMag1FixedClampRS = TRUE THEN
//		tyP0926LifterMagConv.tyCom.tyBitmapMc.usiValueIdx	:= 0;
//	ELSE
//		tyP0926LifterMagConv.tyCom.tyBitmapMc.usiValueIdx	:= 1;
//	END_IF

END_ACTION
```

#### Act_OptP0926Navi.st
```iecst
ACTION Act_OptP0926Navi:

	IF tyP0926LifterMagConv.tyNaviBack.tyBtnBack.bRtCompl = TRUE THEN
		tyP0926LifterMagConv.tyNaviBack.tyBtnBack.bRtCompl		:= FALSE;
		tyP0926LifterMagConv.tyNaviBack.tyBtnBack.bValue		:= FALSE;

		eChgPage		:= UIP0920MtrNPneuCtrl;

	END_IF

END_ACTION
```

#### Act_OptP0926FullMask.st
```iecst
ACTION Act_OptP0926FullMask:

	IF eCurrPage = UIP0926LifterConv THEN

		IF p_tyDI.bEStopSig = FALSE THEN
			p_tyC0002FullMask ACCESS ADR(tyP0926LifterMagConv.tyFullMaskEStop);

		ELSIF p_tyDI.bCoverSWSig = FALSE THEN
			p_tyC0002FullMask ACCESS ADR(tyP0926LifterMagConv.tyFullMaskCWSig);

		ELSIF p_tyDI.bSafetyRlySig = FALSE THEN
			p_tyC0002FullMask ACCESS ADR(tyP0926LifterMagConv.tyFullMaskSafetyRly);

		ELSE
			p_tyC0002FullMask ACCESS ADR(tyP0926LifterMagConv.tyFullMaskHide);

		END_IF

	END_IF

END_ACTION
```

#### Act_OptP0926LifterMagConvChgLyr.st
```iecst
ACTION Act_OptP0926LifterMagConvChgLyr:

	IF tyP0926LifterMagConv.tyCom.tyBtnDCCtrl.bRtCompl THEN
		tyP0926LifterMagConv.tyCom.tyBtnDCCtrl.bRtCompl := FALSE;

		IF tyP0926LifterMagConv.tyCom.tyBtnDCCtrl.bValue = TRUE THEN
			fUIInRtStatOff(ADR(tyP0926LifterMagConv.tyDC.tyLyr.uiRtStat));
			fUIInRtStatHide(ADR(tyP0926LifterMagConv.tyFB.tyLyr.uiRtStat));
		ELSE
			fUIInRtStatHide(ADR(tyP0926LifterMagConv.tyDC.tyLyr.uiRtStat));
			fUIInRtStatOff(ADR(tyP0926LifterMagConv.tyFB.tyLyr.uiRtStat));
		END_IF

	END_IF

END_ACTION
```

#### Act_OptP0926LifterMagConvSen.st
```iecst
ACTION Act_OptP0926LifterMagConvSen:

	tyP0926LifterMagConv.tyCom.tyBtnLifterLmtSW.bValue					:= p_tyDI.bLifterLmtSW;
	tyP0926LifterMagConv.tyCom.tyBtnClampRS.bValue						:= p_tyDI.bMag1FixedClampRS;
	tyP0926LifterMagConv.tyCom.tyBtnUnclampRS.bValue					:= p_tyDI.bMag1FixedUnclampRS;

//	IF p_tyDI.bMag1FixedClampRS = TRUE THEN
//		tyP0926LifterMagConv.tyCom.tyBitmapMc.usiValueIdx	:= 0;
//	ELSE
//		tyP0926LifterMagConv.tyCom.tyBitmapMc.usiValueIdx	:= 1;
//	END_IF

END_ACTION
```

#### Act_OptP0926LifterMagConvFB.st
```iecst
ACTION Act_OptP0926LifterMagConvFB:

	IF tyP0926LifterMagConv.tyFB.tyBtnStop.bRtCompl = TRUE THEN
		eLifterMagConvAct		:= MagConvActStop;

		IF p_eLifterMagConvStat = MagConvActStop AND p_eLifterMagConvStatus = Done THEN
			eLifterMagConvAct	:= MagConvActIdle;

			tyP0926LifterMagConv.tyFB.tyBtnEnter.bRtCompl			:= FALSE;
			tyP0926LifterMagConv.tyFB.tyBtnEnter.bValue				:= FALSE;
			tyP0926LifterMagConv.tyFB.tyBtnEnter.bRtLk				:= FALSE;

			tyP0926LifterMagConv.tyFB.tyBtnExit.bRtCompl			:= FALSE;
			tyP0926LifterMagConv.tyFB.tyBtnExit.bValue				:= FALSE;
			tyP0926LifterMagConv.tyFB.tyBtnExit.bRtLk				:= FALSE;

			tyP0926LifterMagConv.tyFB.tyBtnStop.bRtCompl			:= FALSE;
			tyP0926LifterMagConv.tyFB.tyBtnStop.bValue				:= TRUE;
			tyP0926LifterMagConv.tyFB.tyBtnStop.bRtLk				:= TRUE;
		END_IF

	ELSIF tyP0926LifterMagConv.tyFB.tyBtnEnter.bRtCompl = TRUE THEN
		tyP0926LifterMagConv.tyFB.tyBtnEnter.bValue					:= TRUE;
		tyP0926LifterMagConv.tyFB.tyBtnEnter.bRtLk					:= TRUE;

		tyP0926LifterMagConv.tyFB.tyBtnStop.bValue					:= FALSE;
		tyP0926LifterMagConv.tyFB.tyBtnStop.bRtLk					:= FALSE;

		eLifterMagConvAct		:= MagConvActEnt;

		fUIInRtStatOff(ADR(tyP0926LifterMagConv.tyCom.tyBtnDCCtrl.uiMaskRtStat));

		IF p_eLifterMagConvStat = MagConvActEnt AND p_eLifterMagConvStatus = Done THEN
			eLifterMagConvAct	:= MagConvActIdle;

			tyP0926LifterMagConv.tyFB.tyBtnEnter.bRtCompl			:= FALSE;

			tyP0926LifterMagConv.tyFB.tyBtnEnter.bValue				:= FALSE;
			tyP0926LifterMagConv.tyFB.tyBtnEnter.bRtLk				:= FALSE;

			tyP0926LifterMagConv.tyFB.tyBtnStop.bValue				:= TRUE;
			tyP0926LifterMagConv.tyFB.tyBtnStop.bRtLk				:= TRUE;

			fUIInRtStatHide(ADR(tyP0926LifterMagConv.tyCom.tyBtnDCCtrl.uiMaskRtStat));

		END_IF

	ELSIF tyP0926LifterMagConv.tyFB.tyBtnExit.bRtCompl = TRUE THEN
		tyP0926LifterMagConv.tyFB.tyBtnExit.bValue					:= TRUE;
		tyP0926LifterMagConv.tyFB.tyBtnExit.bRtLk					:= TRUE;

		tyP0926LifterMagConv.tyFB.tyBtnStop.bValue					:= FALSE;
		tyP0926LifterMagConv.tyFB.tyBtnStop.bRtLk					:= FALSE;

		eLifterMagConvAct		:= MagConvActExit;

		fUIInRtStatOff(ADR(tyP0926LifterMagConv.tyCom.tyBtnDCCtrl.uiMaskRtStat));

		IF p_eLifterMagConvStat = MagConvActExit AND p_eLifterMagConvStatus = Done THEN
			eLifterMagConvAct	:= MagConvActIdle;

			tyP0926LifterMagConv.tyFB.tyBtnExit.bRtCompl			:= FALSE;

			tyP0926LifterMagConv.tyFB.tyBtnExit.bValue				:= FALSE;
			tyP0926LifterMagConv.tyFB.tyBtnExit.bRtLk				:= FALSE;

			tyP0926LifterMagConv.tyFB.tyBtnStop.bValue				:= TRUE;
			tyP0926LifterMagConv.tyFB.tyBtnStop.bRtLk				:= TRUE;

			fUIInRtStatHide(ADR(tyP0926LifterMagConv.tyCom.tyBtnDCCtrl.uiMaskRtStat));
		END_IF

	END_IF

	IF tyP0926LifterMagConv.tyCom.tyBtnDCCtrl.bValue = FALSE THEN

		IF tyP0926LifterMagConv.tyFB.tyBtnClamp.bRtCompl = TRUE THEN
			tyP0926LifterMagConv.tyFB.tyBtnClamp.bRtCompl			:= FALSE;

			tyP0926LifterMagConv.tyFB.tyBtnClamp.bValue				:= TRUE;
			tyP0926LifterMagConv.tyFB.tyBtnUnclamp.bValue			:= FALSE;

		ELSIF tyP0926LifterMagConv.tyFB.tyBtnUnclamp.bRtCompl = TRUE THEN
			tyP0926LifterMagConv.tyFB.tyBtnUnclamp.bRtCompl			:= FALSE;

			tyP0926LifterMagConv.tyFB.tyBtnUnclamp.bValue			:= TRUE;
			tyP0926LifterMagConv.tyFB.tyBtnClamp.bValue 			:= FALSE;

		END_IF

		IF tyP0926LifterMagConv.tyFB.tyBtnClamp.bValue = TRUE THEN
			eLifterMagConvAct		:= MagConvActClprClamp;

			IF p_eLifterMagConvStat = MagConvActClprClamp AND p_eLifterMagConvStatus = Done THEN
				eLifterMagConvAct	:= MagConvActIdle;

				tyP0926LifterMagConv.tyFB.tyBtnClamp.bValue			:= FALSE;

			ELSIF p_eLifterMagConvStatus = Error THEN
				tyP0926LifterMagConv.tyFB.tyBtnClamp.bValue			:= FALSE;

			END_IF

		ELSIF tyP0926LifterMagConv.tyFB.tyBtnUnclamp.bValue = TRUE THEN
			eLifterMagConvAct		:= MagConvActClprUnclamp;

			IF p_eLifterMagConvStat = MagConvActClprUnclamp AND p_eLifterMagConvStatus = Done THEN
				eLifterMagConvAct	:= MagConvActIdle;

				tyP0926LifterMagConv.tyFB.tyBtnUnclamp.bValue		:= FALSE;

			ELSIF p_eLifterMagConvStatus = Error THEN
				tyP0926LifterMagConv.tyFB.tyBtnUnclamp.bValue		:= FALSE;

			END_IF

		END_IF

		//Update Status
		tyP0926LifterMagConv.tyDC.tyBtnClamp.bValue					:= p_bLifterMagConvClprClampCtrl;
		tyP0926LifterMagConv.tyDC.tyBtnUnclamp.bValue				:= NOT p_bLifterMagConvClprClampCtrl;

	END_IF

	//Mask
	IF p_tyUsrMgmtCurrAccessRgt.bManualFBOnly THEN
		fUIInRtStatOff(ADR(tyP0926LifterMagConv.tyCom.tyBtnDCCtrl.uiMaskRtStat));

	ELSE

		IF (p_eLifterMagConvStatus = Error) THEN
		fUIInRtStatOff(ADR(tyP0926LifterMagConv.tyFB.tyBtnEnter.uiMaskRtStat));
		fUIInRtStatOff(ADR(tyP0926LifterMagConv.tyFB.tyBtnExit.uiMaskRtStat));
		fUIInRtStatOff(ADR(tyP0926LifterMagConv.tyFB.tyBtnClamp.uiMaskRtStat));
		fUIInRtStatOff(ADR(tyP0926LifterMagConv.tyFB.tyBtnUnclamp.uiMaskRtStat));
		fUIInRtStatHide(ADR(tyP0926LifterMagConv.tyCom.tyBtnDCCtrl.uiMaskRtStat));

		ELSIF tyP0926LifterMagConv.tyFB.tyBtnEnter.bRtCompl = TRUE THEN
		fUIInRtStatHide(ADR(tyP0926LifterMagConv.tyFB.tyBtnEnter.uiMaskRtStat));
		fUIInRtStatOff(ADR(tyP0926LifterMagConv.tyFB.tyBtnExit.uiMaskRtStat));
		fUIInRtStatOff(ADR(tyP0926LifterMagConv.tyFB.tyBtnClamp.uiMaskRtStat));
		fUIInRtStatOff(ADR(tyP0926LifterMagConv.tyFB.tyBtnUnclamp.uiMaskRtStat));
		fUIInRtStatOff(ADR(tyP0926LifterMagConv.tyCom.tyBtnDCCtrl.uiMaskRtStat));

		ELSIF tyP0926LifterMagConv.tyFB.tyBtnExit.bRtCompl = TRUE THEN
		fUIInRtStatOff(ADR(tyP0926LifterMagConv.tyFB.tyBtnEnter.uiMaskRtStat));
		fUIInRtStatHide(ADR(tyP0926LifterMagConv.tyFB.tyBtnExit.uiMaskRtStat));
		fUIInRtStatOff(ADR(tyP0926LifterMagConv.tyFB.tyBtnClamp.uiMaskRtStat));
		fUIInRtStatOff(ADR(tyP0926LifterMagConv.tyFB.tyBtnUnclamp.uiMaskRtStat));
		fUIInRtStatOff(ADR(tyP0926LifterMagConv.tyCom.tyBtnDCCtrl.uiMaskRtStat));

		ELSIF tyP0926LifterMagConv.tyFB.tyBtnClamp.bRtCompl = TRUE OR tyP0926LifterMagConv.tyFB.tyBtnUnclamp.bRtCompl = TRUE THEN
		fUIInRtStatOff(ADR(tyP0926LifterMagConv.tyFB.tyBtnEnter.uiMaskRtStat));
		fUIInRtStatOff(ADR(tyP0926LifterMagConv.tyFB.tyBtnExit.uiMaskRtStat));
		fUIInRtStatHide(ADR(tyP0926LifterMagConv.tyFB.tyBtnClamp.uiMaskRtStat));
		fUIInRtStatHide(ADR(tyP0926LifterMagConv.tyFB.tyBtnUnclamp.uiMaskRtStat));
		fUIInRtStatOff(ADR(tyP0926LifterMagConv.tyCom.tyBtnDCCtrl.uiMaskRtStat));

		ELSE
		fUIInRtStatHide(ADR(tyP0926LifterMagConv.tyFB.tyBtnEnter.uiMaskRtStat));
		fUIInRtStatHide(ADR(tyP0926LifterMagConv.tyFB.tyBtnExit.uiMaskRtStat));
		fUIInRtStatHide(ADR(tyP0926LifterMagConv.tyFB.tyBtnClamp.uiMaskRtStat));
		fUIInRtStatHide(ADR(tyP0926LifterMagConv.tyFB.tyBtnUnclamp.uiMaskRtStat));
		fUIInRtStatHide(ADR(tyP0926LifterMagConv.tyCom.tyBtnDCCtrl.uiMaskRtStat));

		END_IF
	END_IF

END_ACTION
```

#### Act_OptP0926LifterMagConvFBStat.st
```iecst
ACTION Act_OptP0926LifterMagConvFBStat:

	tyP0926LifterMagConv.tyFB.tyStringStat.sValue	:= p_sLifterMagConvStatTxt;

END_ACTION
```

#### Act_OptP0926LifterMagConvDC.st
```iecst
ACTION Act_OptP0926LifterMagConvDC:

	IF tyP0926LifterMagConv.tyDC.tyBtnStop.bRtCompl = TRUE THEN
		tyP0926LifterMagConv.tyDC.tyBtnStop.bValue				:= TRUE;
		tyP0926LifterMagConv.tyDC.tyBtnStop.bRtLk				:= TRUE;

		tyP0926LifterMagConv.tyDC.tyBtnMagIn.bValue				:= FALSE;
		tyP0926LifterMagConv.tyDC.tyBtnMagIn.bRtLk				:= FALSE;

		tyP0926LifterMagConv.tyDC.tyBtnMagOut.bValue			:= FALSE;
		tyP0926LifterMagConv.tyDC.tyBtnMagOut.bRtLk				:= FALSE;

		eLifterMagConvAct		:= MagConvActStop;

		IF p_eLifterMagConvStat = MagConvActStop AND p_eLifterMagConvStatus = Done THEN
			eLifterMagConvAct	:= MagConvActIdle;

			tyP0926LifterMagConv.tyDC.tyBtnStop.bRtCompl		:= FALSE;
		END_IF

	ELSIF tyP0926LifterMagConv.tyDC.tyBtnMagIn.bRtCompl = TRUE THEN
		tyP0926LifterMagConv.tyDC.tyBtnMagIn.bValue				:= TRUE;
		tyP0926LifterMagConv.tyDC.tyBtnMagIn.bRtLk				:= TRUE;

		tyP0926LifterMagConv.tyDC.tyBtnStop.bValue				:= FALSE;
		tyP0926LifterMagConv.tyDC.tyBtnStop.bRtLk				:= FALSE;

		eLifterMagConvAct		:= MagConvActSetMtrDirOrRToL;

		IF p_eLifterMagConvStat = MagConvActSetMtrDirOrRToL AND p_eLifterMagConvStatus = Done THEN

			eLifterMagConvAct	:= MagConvActIdle;

			tyP0926LifterMagConv.tyDC.tyBtnMagIn.bRtCompl		:= FALSE;
		END_IF

	ELSIF tyP0926LifterMagConv.tyDC.tyBtnMagOut.bRtCompl = TRUE THEN

		tyP0926LifterMagConv.tyDC.tyBtnMagOut.bValue			:= TRUE;
		tyP0926LifterMagConv.tyDC.tyBtnMagOut.bRtLk				:= TRUE;

		tyP0926LifterMagConv.tyDC.tyBtnStop.bValue				:= FALSE;
		tyP0926LifterMagConv.tyDC.tyBtnStop.bRtLk				:= FALSE;

		eLifterMagConvAct		:= MagConvActSetMtrSigOnOrLToR;

		IF p_eLifterMagConvStat = MagConvActSetMtrSigOnOrLToR AND p_eLifterMagConvStatus = Done THEN

			eLifterMagConvAct	:= MagConvActIdle;

			tyP0926LifterMagConv.tyDC.tyBtnMagOut.bRtCompl		:= FALSE;
		END_IF

	END_IF

	//Clamper
	IF p_bLifterMagConvClprTwoCtrlOut = FALSE THEN
		IF tyP0926LifterMagConv.tyDC.tyBtnClamp.bRtCompl = TRUE THEN
			tyP0926LifterMagConv.tyDC.tyBtnClamp.bValue			:= TRUE;
			tyP0926LifterMagConv.tyDC.tyBtnUnclamp.bValue		:= FALSE;

			eLifterMagConvAct		:= MagConvActClprSetClamp;

			IF p_eLifterMagConvStat = MagConvActClprSetClamp AND p_eLifterMagConvStatus = Done THEN
				eLifterMagConvAct	:= MagConvActIdle;

				tyP0926LifterMagConv.tyDC.tyBtnClamp.bRtCompl	:= FALSE;
			END_IF

		ELSIF tyP0926LifterMagConv.tyDC.tyBtnUnclamp.bRtCompl = TRUE THEN
			tyP0926LifterMagConv.tyDC.tyBtnUnclamp.bValue		:= TRUE;
			tyP0926LifterMagConv.tyDC.tyBtnClamp.bValue			:= FALSE;

			eLifterMagConvAct		:= MagConvActClprSetUnclamp;

			IF p_eLifterMagConvStat = MagConvActClprSetUnclamp AND p_eLifterMagConvStatus = Done THEN
				eLifterMagConvAct	:= MagConvActIdle;

				tyP0926LifterMagConv.tyDC.tyBtnUnclamp.bRtCompl	:= FALSE;
			END_IF
		END_IF

	ELSE
		IF (tyP0926LifterMagConv.tyDC.tyBtnClamp.bRtCompl = TRUE) OR (tyP0926LifterMagConv.tyDC.tyBtnUnclamp.bRtCompl = TRUE) THEN
			IF (tyP0926LifterMagConv.tyDC.tyBtnClamp.bValue = TRUE) AND (tyP0926LifterMagConv.tyDC.tyBtnUnclamp.bValue = TRUE) THEN

				eLifterMagConvAct	:= MagConvActClprSetAll;

				IF p_eLifterMagConvStat = MagConvActClprSetAll AND p_eLifterMagConvStatus = Done THEN
					eLifterMagConvAct	:= MagConvActIdle;

					tyP0926LifterMagConv.tyDC.tyBtnClamp.bRtCompl	:= FALSE;
					tyP0926LifterMagConv.tyDC.tyBtnUnclamp.bRtCompl	:= FALSE;
				END_IF

			ELSIF (tyP0926LifterMagConv.tyDC.tyBtnClamp.bValue = TRUE) AND (tyP0926LifterMagConv.tyDC.tyBtnUnclamp.bValue = FALSE) THEN

				eLifterMagConvAct		:= MagConvActClprSetClamp;

				IF p_eLifterMagConvStat = MagConvActClprSetClamp AND p_eLifterMagConvStatus = Done THEN

					eLifterMagConvAct	:= MagConvActIdle;

					tyP0926LifterMagConv.tyDC.tyBtnClamp.bRtCompl	:= FALSE;
					tyP0926LifterMagConv.tyDC.tyBtnUnclamp.bRtCompl	:= FALSE;
				END_IF

			ELSIF (tyP0926LifterMagConv.tyDC.tyBtnClamp.bValue = FALSE) AND (tyP0926LifterMagConv.tyDC.tyBtnUnclamp.bValue = TRUE) THEN

				eLifterMagConvAct		:= MagConvActClprSetUnclamp;

				IF p_eLifterMagConvStat = MagConvActClprSetUnclamp AND p_eLifterMagConvStatus = Done THEN

					eLifterMagConvAct	:= MagConvActIdle;

					tyP0926LifterMagConv.tyDC.tyBtnClamp.bRtCompl	:= FALSE;
					tyP0926LifterMagConv.tyDC.tyBtnUnclamp.bRtCompl	:= FALSE;
				END_IF

			ELSE
				eLifterMagConvAct		:= MagConvActClprRstAll;

				IF p_eLifterMagConvStat = MagConvActClprRstAll AND p_eLifterMagConvStatus = Done THEN

					eLifterMagConvAct	:= MagConvActIdle;

					tyP0926LifterMagConv.tyDC.tyBtnClamp.bRtCompl	:= FALSE;
					tyP0926LifterMagConv.tyDC.tyBtnUnclamp.bRtCompl	:= FALSE;
				END_IF

			END_IF
		END_IF
	END_IF

	IF tyP0926LifterMagConv.tyCom.tyBtnDCCtrl.bValue = TRUE THEN
		tyP0926LifterMagConv.tyFB.tyBtnClamp.bRtCompl				:= FALSE;
		tyP0926LifterMagConv.tyFB.tyBtnUnclamp.bRtCompl				:= FALSE;
		tyP0926LifterMagConv.tyFB.tyBtnClamp.bValue					:= FALSE;
		tyP0926LifterMagConv.tyFB.tyBtnUnclamp.bValue				:= FALSE;
	END_IF

	//Mask

	IF p_eLifterMagConvStatus = Error THEN
		fUIInRtStatOff(ADR(tyP0926LifterMagConv.tyDC.tyBtnMagIn.uiMaskRtStat));
		fUIInRtStatOff(ADR(tyP0926LifterMagConv.tyDC.tyBtnMagOut.uiMaskRtStat));
		fUIInRtStatOff(ADR(tyP0926LifterMagConv.tyDC.tyBtnClamp.uiMaskRtStat));
		fUIInRtStatOff(ADR(tyP0926LifterMagConv.tyDC.tyBtnUnclamp.uiMaskRtStat));

	ELSIF tyP0926LifterMagConv.tyDC.tyBtnMagIn.bRtCompl = TRUE THEN
		fUIInRtStatHide(ADR(tyP0926LifterMagConv.tyDC.tyBtnMagIn.uiMaskRtStat));
		fUIInRtStatOff(ADR(tyP0926LifterMagConv.tyDC.tyBtnMagOut.uiMaskRtStat));
		fUIInRtStatOff(ADR(tyP0926LifterMagConv.tyDC.tyBtnClamp.uiMaskRtStat));
		fUIInRtStatOff(ADR(tyP0926LifterMagConv.tyDC.tyBtnUnclamp.uiMaskRtStat));

	ELSIF tyP0926LifterMagConv.tyDC.tyBtnMagOut.bRtCompl = TRUE THEN
		fUIInRtStatOff(ADR(tyP0926LifterMagConv.tyDC.tyBtnMagIn.uiMaskRtStat));
		fUIInRtStatHide(ADR(tyP0926LifterMagConv.tyDC.tyBtnMagOut.uiMaskRtStat));
		fUIInRtStatOff(ADR(tyP0926LifterMagConv.tyDC.tyBtnClamp.uiMaskRtStat));
		fUIInRtStatOff(ADR(tyP0926LifterMagConv.tyDC.tyBtnUnclamp.uiMaskRtStat));

	ELSIF tyP0926LifterMagConv.tyDC.tyBtnStop.bRtCompl = TRUE THEN
		fUIInRtStatHide(ADR(tyP0926LifterMagConv.tyDC.tyBtnMagIn.uiMaskRtStat));
		fUIInRtStatHide(ADR(tyP0926LifterMagConv.tyDC.tyBtnMagOut.uiMaskRtStat));
		fUIInRtStatHide(ADR(tyP0926LifterMagConv.tyDC.tyBtnClamp.uiMaskRtStat));
		fUIInRtStatHide(ADR(tyP0926LifterMagConv.tyDC.tyBtnUnclamp.uiMaskRtStat));

	END_IF

END_ACTION
```

#### Act_OptP0926RstMnl.st
```iecst
ACTION Act_OptP0926RstMnl:

	IF EDGEPOS((bManualMod = FALSE) OR (p_eLifterMagConvStatus = Error)) THEN

		eLifterMagConvAct	:= MagConvActIdle;

		//Lifter Mag Conveyor
		//FB
		tyP0926LifterMagConv.tyFB.tyBtnEnter.bRtCompl				:= FALSE;
		tyP0926LifterMagConv.tyFB.tyBtnExit.bRtCompl				:= FALSE;
		tyP0926LifterMagConv.tyFB.tyBtnStop.bRtCompl				:= FALSE;

		tyP0926LifterMagConv.tyFB.tyBtnEnter.bValue					:= FALSE;
		tyP0926LifterMagConv.tyFB.tyBtnExit.bValue					:= FALSE;
		tyP0926LifterMagConv.tyFB.tyBtnStop.bValue					:= TRUE;

		tyP0926LifterMagConv.tyFB.tyBtnEnter.bRtLk					:= FALSE;
		tyP0926LifterMagConv.tyFB.tyBtnExit.bRtLk					:= FALSE;
		tyP0926LifterMagConv.tyFB.tyBtnStop.bRtLk					:= TRUE;

		tyP0926LifterMagConv.tyFB.tyBtnEnter.uiMaskRtStat.0			:= TRUE;
		tyP0926LifterMagConv.tyFB.tyBtnExit.uiMaskRtStat.0			:= TRUE;
		tyP0926LifterMagConv.tyCom.tyBtnDCCtrl.uiMaskRtStat.0		:= TRUE;

		//Direct
		tyP0926LifterMagConv.tyDC.tyBtnMagIn.bRtCompl				:= FALSE;
		tyP0926LifterMagConv.tyDC.tyBtnMagOut.bRtCompl				:= FALSE;
		tyP0926LifterMagConv.tyDC.tyBtnStop.bRtCompl				:= FALSE;

		tyP0926LifterMagConv.tyDC.tyBtnMagIn.bValue					:= FALSE;
		tyP0926LifterMagConv.tyDC.tyBtnMagOut.bValue				:= FALSE;
		tyP0926LifterMagConv.tyDC.tyBtnStop.bValue					:= TRUE;

		tyP0926LifterMagConv.tyDC.tyBtnMagIn.bRtLk					:= FALSE;
		tyP0926LifterMagConv.tyDC.tyBtnMagOut.bRtLk					:= FALSE;
		tyP0926LifterMagConv.tyDC.tyBtnStop.bRtLk					:= TRUE;

		tyP0926LifterMagConv.tyDC.tyBtnMagIn.uiMaskRtStat.0			:= TRUE;
		tyP0926LifterMagConv.tyDC.tyBtnMagOut.uiMaskRtStat.0		:= TRUE;
		tyP0926LifterMagConv.tyCom.tyBtnDCCtrl.uiMaskRtStat.0		:= TRUE;

		//Mag Clamper
		//FB
		tyP0926LifterMagConv.tyFB.tyBtnClamp.bRtCompl				:= FALSE;
		tyP0926LifterMagConv.tyFB.tyBtnUnclamp.bRtCompl				:= FALSE;

		tyP0926LifterMagConv.tyFB.tyBtnClamp.bValue					:= FALSE;
		tyP0926LifterMagConv.tyFB.tyBtnUnclamp.bValue				:= FALSE;

		tyP0926LifterMagConv.tyFB.tyBtnClamp.uiMaskRtStat.0			:= TRUE;
		tyP0926LifterMagConv.tyFB.tyBtnUnclamp.uiMaskRtStat.0		:= TRUE;
		tyP0926LifterMagConv.tyCom.tyBtnDCCtrl.uiMaskRtStat.0		:= TRUE;

		//Direct
		tyP0926LifterMagConv.tyDC.tyBtnClamp.bRtCompl				:= FALSE;
		tyP0926LifterMagConv.tyDC.tyBtnUnclamp.bRtCompl				:= FALSE;

		tyP0926LifterMagConv.tyDC.tyBtnClamp.bValue					:= FALSE;
		tyP0926LifterMagConv.tyDC.tyBtnUnclamp.bValue				:= FALSE;

		tyP0926LifterMagConv.tyDC.tyBtnClamp.uiMaskRtStat.0			:= TRUE;
		tyP0926LifterMagConv.tyDC.tyBtnUnclamp.uiMaskRtStat.0		:= TRUE;
		tyP0926LifterMagConv.tyCom.tyBtnDCCtrl.uiMaskRtStat.0		:= TRUE;

	END_IF

	IF EDGEPOS(bManualMod = FALSE) THEN

		tyP0926LifterMagConv.tyCom.tyBtnDCCtrl.bValue	:= FALSE;

		fUIInRtStatOff(ADR(tyP0926LifterMagConv.tyFB.tyLyr.uiRtStat));
		fUIInRtStatHide(ADR(tyP0926LifterMagConv.tyDC.tyLyr.uiRtStat));

	END_IF

END_ACTION
```

#### Act_EntP0927Disp.st
```iecst
ACTION Act_EntP0927Disp:

	// Access Address
	p_tyC0002FullMask ACCESS ADR(tyP0927LifterMagConv2.tyFullMaskHide);

	p_tyC0004Navi ACCESS ADR(tyP0927LifterMagConv2.tyNaviBack);

	p_tyC0005Main ACCESS ADR(tyCommon.tyMain);

	p_tyC0007Notif ACCESS ADR(tyCommon.tyNotif);

	p_tyC0008MsgBox ACCESS ADR(tyP0927LifterMagConv2.tyMsgBoxHide);

	p_tyC0009Info ACCESS ADR(tyCommon.tyInfo);

	p_tyP0927LifterMagConvCom ACCESS ADR(tyP0927LifterMagConv2.tyCom);
	p_tyP0927LifterMagConvDC ACCESS ADR(tyP0927LifterMagConv2.tyDC);
	p_tyP0927LifterMagConvFB ACCESS ADR(tyP0927LifterMagConv2.tyFB);

	// Display
//	IF p_tyDI.bMag1FixedClampRS = TRUE THEN
//		tyP0927LifterMagConv2.tyCom.tyBitmapMc.usiValueIdx	:= 0;
//	ELSE
//		tyP0927LifterMagConv2.tyCom.tyBitmapMc.usiValueIdx	:= 1;
//	END_IF

END_ACTION
```

#### Act_OptP0927Navi.st
```iecst
ACTION Act_OptP0927Navi:

	IF tyP0927LifterMagConv2.tyNaviBack.tyBtnBack.bRtCompl = TRUE THEN
		tyP0927LifterMagConv2.tyNaviBack.tyBtnBack.bRtCompl		:= FALSE;
		tyP0927LifterMagConv2.tyNaviBack.tyBtnBack.bValue		:= FALSE;

		eChgPage		:= UIP0920MtrNPneuCtrl;

	END_IF

END_ACTION
```

#### Act_OptP0927FullMask.st
```iecst
ACTION Act_OptP0927FullMask:

	IF eCurrPage = UIP0927LifterConv2 THEN

		IF p_tyDI.bEStopSig = FALSE THEN
			p_tyC0002FullMask ACCESS ADR(tyP0927LifterMagConv2.tyFullMaskEStop);

		ELSIF p_tyDI.bCoverSWSig = FALSE THEN
			p_tyC0002FullMask ACCESS ADR(tyP0927LifterMagConv2.tyFullMaskCWSig);

		ELSIF p_tyDI.bSafetyRlySig = FALSE THEN
			p_tyC0002FullMask ACCESS ADR(tyP0927LifterMagConv2.tyFullMaskSafetyRly);

		ELSE
			p_tyC0002FullMask ACCESS ADR(tyP0927LifterMagConv2.tyFullMaskHide);

		END_IF

	END_IF

END_ACTION
```

#### Act_OptP0927LifterMagConvChgLyr.st
```iecst
ACTION Act_OptP0927LifterMagConvChgLyr:

	IF tyP0927LifterMagConv2.tyCom.tyBtnDCCtrl.bRtCompl THEN
		tyP0927LifterMagConv2.tyCom.tyBtnDCCtrl.bRtCompl := FALSE;

		IF tyP0927LifterMagConv2.tyCom.tyBtnDCCtrl.bValue = TRUE THEN
			fUIInRtStatOff(ADR(tyP0927LifterMagConv2.tyDC.tyLyr.uiRtStat));
			fUIInRtStatHide(ADR(tyP0927LifterMagConv2.tyFB.tyLyr.uiRtStat));
		ELSE
			fUIInRtStatHide(ADR(tyP0927LifterMagConv2.tyDC.tyLyr.uiRtStat));
			fUIInRtStatOff(ADR(tyP0927LifterMagConv2.tyFB.tyLyr.uiRtStat));
		END_IF

	END_IF

END_ACTION
```

#### Act_OptP0927LifterMagConvSen.st
```iecst
ACTION Act_OptP0927LifterMagConvSen:

	tyP0927LifterMagConv2.tyCom.tyBtnLifterLmtSW.bValue					:= p_tyDI.bLifter2LmtSW;
	tyP0927LifterMagConv2.tyCom.tyBtnClampRS.bValue						:= p_tyDI.bMag2FixedClampRS;
	tyP0927LifterMagConv2.tyCom.tyBtnUnclampRS.bValue					:= p_tyDI.bMag2FixedUnclampRS;

//	IF p_tyDI.bMag2FixedClampRS = TRUE THEN
//		tyP0927LifterMagConv2.tyCom.tyBitmapMc.usiValueIdx	:= 0;
//	ELSE
//		tyP0927LifterMagConv2.tyCom.tyBitmapMc.usiValueIdx	:= 1;
//	END_IF

END_ACTION
```

#### Act_OptP0927LifterMagConvFB.st
```iecst
ACTION Act_OptP0927LifterMagConvFB:

	IF tyP0927LifterMagConv2.tyFB.tyBtnStop.bRtCompl = TRUE THEN
		eLifterMagConv2Act		:= MagConvActStop;

		IF p_eLifterMagConv2Stat = MagConvActStop AND p_eLifterMagConv2Status = Done THEN
			eLifterMagConv2Act	:= MagConvActIdle;

			tyP0927LifterMagConv2.tyFB.tyBtnEnter.bRtCompl			:= FALSE;
			tyP0927LifterMagConv2.tyFB.tyBtnEnter.bValue				:= FALSE;
			tyP0927LifterMagConv2.tyFB.tyBtnEnter.bRtLk				:= FALSE;

			tyP0927LifterMagConv2.tyFB.tyBtnExit.bRtCompl			:= FALSE;
			tyP0927LifterMagConv2.tyFB.tyBtnExit.bValue				:= FALSE;
			tyP0927LifterMagConv2.tyFB.tyBtnExit.bRtLk				:= FALSE;

			tyP0927LifterMagConv2.tyFB.tyBtnStop.bRtCompl			:= FALSE;
			tyP0927LifterMagConv2.tyFB.tyBtnStop.bValue				:= TRUE;
			tyP0927LifterMagConv2.tyFB.tyBtnStop.bRtLk				:= TRUE;
		END_IF

	ELSIF tyP0927LifterMagConv2.tyFB.tyBtnEnter.bRtCompl = TRUE THEN
		tyP0927LifterMagConv2.tyFB.tyBtnEnter.bValue					:= TRUE;
		tyP0927LifterMagConv2.tyFB.tyBtnEnter.bRtLk					:= TRUE;

		tyP0927LifterMagConv2.tyFB.tyBtnStop.bValue					:= FALSE;
		tyP0927LifterMagConv2.tyFB.tyBtnStop.bRtLk					:= FALSE;

		eLifterMagConv2Act		:= MagConvActEnt;

		fUIInRtStatOff(ADR(tyP0927LifterMagConv2.tyCom.tyBtnDCCtrl.uiMaskRtStat));

		IF p_eLifterMagConv2Stat = MagConvActEnt AND p_eLifterMagConv2Status = Done THEN
			eLifterMagConv2Act	:= MagConvActIdle;

			tyP0927LifterMagConv2.tyFB.tyBtnEnter.bRtCompl			:= FALSE;

			tyP0927LifterMagConv2.tyFB.tyBtnEnter.bValue				:= FALSE;
			tyP0927LifterMagConv2.tyFB.tyBtnEnter.bRtLk				:= FALSE;

			tyP0927LifterMagConv2.tyFB.tyBtnStop.bValue				:= TRUE;
			tyP0927LifterMagConv2.tyFB.tyBtnStop.bRtLk				:= TRUE;

			fUIInRtStatHide(ADR(tyP0927LifterMagConv2.tyCom.tyBtnDCCtrl.uiMaskRtStat));

		END_IF

	ELSIF tyP0927LifterMagConv2.tyFB.tyBtnExit.bRtCompl = TRUE THEN
		tyP0927LifterMagConv2.tyFB.tyBtnExit.bValue					:= TRUE;
		tyP0927LifterMagConv2.tyFB.tyBtnExit.bRtLk					:= TRUE;

		tyP0927LifterMagConv2.tyFB.tyBtnStop.bValue					:= FALSE;
		tyP0927LifterMagConv2.tyFB.tyBtnStop.bRtLk					:= FALSE;

		eLifterMagConv2Act		:= MagConvActExit;

		fUIInRtStatOff(ADR(tyP0927LifterMagConv2.tyCom.tyBtnDCCtrl.uiMaskRtStat));

		IF p_eLifterMagConv2Stat = MagConvActExit AND p_eLifterMagConv2Status = Done THEN
			eLifterMagConv2Act	:= MagConvActIdle;

			tyP0927LifterMagConv2.tyFB.tyBtnExit.bRtCompl			:= FALSE;

			tyP0927LifterMagConv2.tyFB.tyBtnExit.bValue				:= FALSE;
			tyP0927LifterMagConv2.tyFB.tyBtnExit.bRtLk				:= FALSE;

			tyP0927LifterMagConv2.tyFB.tyBtnStop.bValue				:= TRUE;
			tyP0927LifterMagConv2.tyFB.tyBtnStop.bRtLk				:= TRUE;

			fUIInRtStatHide(ADR(tyP0927LifterMagConv2.tyCom.tyBtnDCCtrl.uiMaskRtStat));
		END_IF

	END_IF

	IF tyP0927LifterMagConv2.tyCom.tyBtnDCCtrl.bValue = FALSE THEN

		IF tyP0927LifterMagConv2.tyFB.tyBtnClamp.bRtCompl = TRUE THEN
			tyP0927LifterMagConv2.tyFB.tyBtnClamp.bRtCompl			:= FALSE;

			tyP0927LifterMagConv2.tyFB.tyBtnClamp.bValue				:= TRUE;
			tyP0927LifterMagConv2.tyFB.tyBtnUnclamp.bValue			:= FALSE;

		ELSIF tyP0927LifterMagConv2.tyFB.tyBtnUnclamp.bRtCompl = TRUE THEN
			tyP0927LifterMagConv2.tyFB.tyBtnUnclamp.bRtCompl			:= FALSE;

			tyP0927LifterMagConv2.tyFB.tyBtnUnclamp.bValue			:= TRUE;
			tyP0927LifterMagConv2.tyFB.tyBtnClamp.bValue 			:= FALSE;

		END_IF

		IF tyP0927LifterMagConv2.tyFB.tyBtnClamp.bValue = TRUE THEN
			eLifterMagConv2Act		:= MagConvActClprClamp;

			IF p_eLifterMagConv2Stat = MagConvActClprClamp AND p_eLifterMagConv2Status = Done THEN
				eLifterMagConv2Act	:= MagConvActIdle;

				tyP0927LifterMagConv2.tyFB.tyBtnClamp.bValue			:= FALSE;

			ELSIF p_eLifterMagConv2Status = Error THEN
				tyP0927LifterMagConv2.tyFB.tyBtnClamp.bValue			:= FALSE;

			END_IF

		ELSIF tyP0927LifterMagConv2.tyFB.tyBtnUnclamp.bValue = TRUE THEN
			eLifterMagConv2Act		:= MagConvActClprUnclamp;

			IF p_eLifterMagConv2Stat = MagConvActClprUnclamp AND p_eLifterMagConv2Status = Done THEN
				eLifterMagConv2Act	:= MagConvActIdle;

				tyP0927LifterMagConv2.tyFB.tyBtnUnclamp.bValue		:= FALSE;

			ELSIF p_eLifterMagConv2Status = Error THEN
				tyP0927LifterMagConv2.tyFB.tyBtnUnclamp.bValue		:= FALSE;

			END_IF

		END_IF

		//Update Status
		tyP0927LifterMagConv2.tyDC.tyBtnClamp.bValue					:= p_bLifterMagConvClprClampCtrl;
		tyP0927LifterMagConv2.tyDC.tyBtnUnclamp.bValue				:= NOT p_bLifterMagConvClprClampCtrl;

	END_IF

	//Mask
	IF p_tyUsrMgmtCurrAccessRgt.bManualFBOnly THEN
		fUIInRtStatOff(ADR(tyP0927LifterMagConv2.tyCom.tyBtnDCCtrl.uiMaskRtStat));

	ELSE

		IF (p_eLifterMagConv2Status = Error) THEN
		fUIInRtStatOff(ADR(tyP0927LifterMagConv2.tyFB.tyBtnEnter.uiMaskRtStat));
		fUIInRtStatOff(ADR(tyP0927LifterMagConv2.tyFB.tyBtnExit.uiMaskRtStat));
		fUIInRtStatOff(ADR(tyP0927LifterMagConv2.tyFB.tyBtnClamp.uiMaskRtStat));
		fUIInRtStatOff(ADR(tyP0927LifterMagConv2.tyFB.tyBtnUnclamp.uiMaskRtStat));
		fUIInRtStatHide(ADR(tyP0927LifterMagConv2.tyCom.tyBtnDCCtrl.uiMaskRtStat));

		ELSIF tyP0927LifterMagConv2.tyFB.tyBtnEnter.bRtCompl = TRUE THEN
		fUIInRtStatHide(ADR(tyP0927LifterMagConv2.tyFB.tyBtnEnter.uiMaskRtStat));
		fUIInRtStatOff(ADR(tyP0927LifterMagConv2.tyFB.tyBtnExit.uiMaskRtStat));
		fUIInRtStatOff(ADR(tyP0927LifterMagConv2.tyFB.tyBtnClamp.uiMaskRtStat));
		fUIInRtStatOff(ADR(tyP0927LifterMagConv2.tyFB.tyBtnUnclamp.uiMaskRtStat));
		fUIInRtStatOff(ADR(tyP0927LifterMagConv2.tyCom.tyBtnDCCtrl.uiMaskRtStat));

		ELSIF tyP0927LifterMagConv2.tyFB.tyBtnExit.bRtCompl = TRUE THEN
		fUIInRtStatOff(ADR(tyP0927LifterMagConv2.tyFB.tyBtnEnter.uiMaskRtStat));
		fUIInRtStatHide(ADR(tyP0927LifterMagConv2.tyFB.tyBtnExit.uiMaskRtStat));
		fUIInRtStatOff(ADR(tyP0927LifterMagConv2.tyFB.tyBtnClamp.uiMaskRtStat));
		fUIInRtStatOff(ADR(tyP0927LifterMagConv2.tyFB.tyBtnUnclamp.uiMaskRtStat));
		fUIInRtStatOff(ADR(tyP0927LifterMagConv2.tyCom.tyBtnDCCtrl.uiMaskRtStat));

		ELSIF tyP0927LifterMagConv2.tyFB.tyBtnClamp.bRtCompl = TRUE OR tyP0927LifterMagConv2.tyFB.tyBtnUnclamp.bRtCompl = TRUE THEN
		fUIInRtStatOff(ADR(tyP0927LifterMagConv2.tyFB.tyBtnEnter.uiMaskRtStat));
		fUIInRtStatOff(ADR(tyP0927LifterMagConv2.tyFB.tyBtnExit.uiMaskRtStat));
		fUIInRtStatHide(ADR(tyP0927LifterMagConv2.tyFB.tyBtnClamp.uiMaskRtStat));
		fUIInRtStatHide(ADR(tyP0927LifterMagConv2.tyFB.tyBtnUnclamp.uiMaskRtStat));
		fUIInRtStatOff(ADR(tyP0927LifterMagConv2.tyCom.tyBtnDCCtrl.uiMaskRtStat));

		ELSE
		fUIInRtStatHide(ADR(tyP0927LifterMagConv2.tyFB.tyBtnEnter.uiMaskRtStat));
		fUIInRtStatHide(ADR(tyP0927LifterMagConv2.tyFB.tyBtnExit.uiMaskRtStat));
		fUIInRtStatHide(ADR(tyP0927LifterMagConv2.tyFB.tyBtnClamp.uiMaskRtStat));
		fUIInRtStatHide(ADR(tyP0927LifterMagConv2.tyFB.tyBtnUnclamp.uiMaskRtStat));
		fUIInRtStatHide(ADR(tyP0927LifterMagConv2.tyCom.tyBtnDCCtrl.uiMaskRtStat));

		END_IF
	END_IF

END_ACTION
```

#### Act_OptP0927LifterMagConvFBStat.st
```iecst
ACTION Act_OptP0927LifterMagConvFBStat:

	tyP0927LifterMagConv2.tyFB.tyStringStat.sValue	:= p_sLifterMagConv2StatTxt;

END_ACTION
```

#### Act_OptP0927LifterMagConvDC.st
```iecst
ACTION Act_OptP0927LifterMagConvDC:

	IF tyP0927LifterMagConv2.tyDC.tyBtnStop.bRtCompl = TRUE THEN
		tyP0927LifterMagConv2.tyDC.tyBtnStop.bValue				:= TRUE;
		tyP0927LifterMagConv2.tyDC.tyBtnStop.bRtLk				:= TRUE;

		tyP0927LifterMagConv2.tyDC.tyBtnMagIn.bValue				:= FALSE;
		tyP0927LifterMagConv2.tyDC.tyBtnMagIn.bRtLk				:= FALSE;

		tyP0927LifterMagConv2.tyDC.tyBtnMagOut.bValue			:= FALSE;
		tyP0927LifterMagConv2.tyDC.tyBtnMagOut.bRtLk				:= FALSE;

		eLifterMagConv2Act		:= MagConvActStop;

		IF p_eLifterMagConv2Stat = MagConvActStop AND p_eLifterMagConv2Status = Done THEN
			eLifterMagConv2Act	:= MagConvActIdle;

			tyP0927LifterMagConv2.tyDC.tyBtnStop.bRtCompl		:= FALSE;
		END_IF

	ELSIF tyP0927LifterMagConv2.tyDC.tyBtnMagIn.bRtCompl = TRUE THEN
		tyP0927LifterMagConv2.tyDC.tyBtnMagIn.bValue				:= TRUE;
		tyP0927LifterMagConv2.tyDC.tyBtnMagIn.bRtLk				:= TRUE;

		tyP0927LifterMagConv2.tyDC.tyBtnStop.bValue				:= FALSE;
		tyP0927LifterMagConv2.tyDC.tyBtnStop.bRtLk				:= FALSE;

		eLifterMagConv2Act		:= MagConvActSetMtrDirOrRToL;

		IF p_eLifterMagConv2Stat = MagConvActSetMtrDirOrRToL AND p_eLifterMagConv2Status = Done THEN

			eLifterMagConv2Act	:= MagConvActIdle;

			tyP0927LifterMagConv2.tyDC.tyBtnMagIn.bRtCompl		:= FALSE;
		END_IF

	ELSIF tyP0927LifterMagConv2.tyDC.tyBtnMagOut.bRtCompl = TRUE THEN

		tyP0927LifterMagConv2.tyDC.tyBtnMagOut.bValue			:= TRUE;
		tyP0927LifterMagConv2.tyDC.tyBtnMagOut.bRtLk				:= TRUE;

		tyP0927LifterMagConv2.tyDC.tyBtnStop.bValue				:= FALSE;
		tyP0927LifterMagConv2.tyDC.tyBtnStop.bRtLk				:= FALSE;

		eLifterMagConv2Act		:= MagConvActSetMtrSigOnOrLToR;

		IF p_eLifterMagConv2Stat = MagConvActSetMtrSigOnOrLToR AND p_eLifterMagConv2Status = Done THEN

			eLifterMagConv2Act	:= MagConvActIdle;

			tyP0927LifterMagConv2.tyDC.tyBtnMagOut.bRtCompl		:= FALSE;
		END_IF

	END_IF

	//Clamper
	IF p_bLifterMagConvClprTwoCtrlOut = FALSE THEN
		IF tyP0927LifterMagConv2.tyDC.tyBtnClamp.bRtCompl = TRUE THEN
			tyP0927LifterMagConv2.tyDC.tyBtnClamp.bValue			:= TRUE;
			tyP0927LifterMagConv2.tyDC.tyBtnUnclamp.bValue		:= FALSE;

			eLifterMagConv2Act		:= MagConvActClprSetClamp;

			IF p_eLifterMagConv2Stat = MagConvActClprSetClamp AND p_eLifterMagConv2Status = Done THEN
				eLifterMagConv2Act	:= MagConvActIdle;

				tyP0927LifterMagConv2.tyDC.tyBtnClamp.bRtCompl	:= FALSE;
			END_IF

		ELSIF tyP0927LifterMagConv2.tyDC.tyBtnUnclamp.bRtCompl = TRUE THEN
			tyP0927LifterMagConv2.tyDC.tyBtnUnclamp.bValue		:= TRUE;
			tyP0927LifterMagConv2.tyDC.tyBtnClamp.bValue			:= FALSE;

			eLifterMagConv2Act		:= MagConvActClprSetUnclamp;

			IF p_eLifterMagConv2Stat = MagConvActClprSetUnclamp AND p_eLifterMagConv2Status = Done THEN
				eLifterMagConv2Act	:= MagConvActIdle;

				tyP0927LifterMagConv2.tyDC.tyBtnUnclamp.bRtCompl	:= FALSE;
			END_IF
		END_IF

	ELSE
		IF (tyP0927LifterMagConv2.tyDC.tyBtnClamp.bRtCompl = TRUE) OR (tyP0927LifterMagConv2.tyDC.tyBtnUnclamp.bRtCompl = TRUE) THEN
			IF (tyP0927LifterMagConv2.tyDC.tyBtnClamp.bValue = TRUE) AND (tyP0927LifterMagConv2.tyDC.tyBtnUnclamp.bValue = TRUE) THEN

				eLifterMagConv2Act	:= MagConvActClprSetAll;

				IF p_eLifterMagConv2Stat = MagConvActClprSetAll AND p_eLifterMagConv2Status = Done THEN
					eLifterMagConv2Act	:= MagConvActIdle;

					tyP0927LifterMagConv2.tyDC.tyBtnClamp.bRtCompl	:= FALSE;
					tyP0927LifterMagConv2.tyDC.tyBtnUnclamp.bRtCompl	:= FALSE;
				END_IF

			ELSIF (tyP0927LifterMagConv2.tyDC.tyBtnClamp.bValue = TRUE) AND (tyP0927LifterMagConv2.tyDC.tyBtnUnclamp.bValue = FALSE) THEN

				eLifterMagConv2Act		:= MagConvActClprSetClamp;

				IF p_eLifterMagConv2Stat = MagConvActClprSetClamp AND p_eLifterMagConv2Status = Done THEN

					eLifterMagConv2Act	:= MagConvActIdle;

					tyP0927LifterMagConv2.tyDC.tyBtnClamp.bRtCompl	:= FALSE;
					tyP0927LifterMagConv2.tyDC.tyBtnUnclamp.bRtCompl	:= FALSE;
				END_IF

			ELSIF (tyP0927LifterMagConv2.tyDC.tyBtnClamp.bValue = FALSE) AND (tyP0927LifterMagConv2.tyDC.tyBtnUnclamp.bValue = TRUE) THEN

				eLifterMagConv2Act		:= MagConvActClprSetUnclamp;

				IF p_eLifterMagConv2Stat = MagConvActClprSetUnclamp AND p_eLifterMagConv2Status = Done THEN

					eLifterMagConv2Act	:= MagConvActIdle;

					tyP0927LifterMagConv2.tyDC.tyBtnClamp.bRtCompl	:= FALSE;
					tyP0927LifterMagConv2.tyDC.tyBtnUnclamp.bRtCompl	:= FALSE;
				END_IF

			ELSE
				eLifterMagConv2Act		:= MagConvActClprRstAll;

				IF p_eLifterMagConv2Stat = MagConvActClprRstAll AND p_eLifterMagConv2Status = Done THEN

					eLifterMagConv2Act	:= MagConvActIdle;

					tyP0927LifterMagConv2.tyDC.tyBtnClamp.bRtCompl	:= FALSE;
					tyP0927LifterMagConv2.tyDC.tyBtnUnclamp.bRtCompl	:= FALSE;
				END_IF

			END_IF
		END_IF
	END_IF

	IF tyP0927LifterMagConv2.tyCom.tyBtnDCCtrl.bValue = TRUE THEN
		tyP0927LifterMagConv2.tyFB.tyBtnClamp.bRtCompl				:= FALSE;
		tyP0927LifterMagConv2.tyFB.tyBtnUnclamp.bRtCompl				:= FALSE;
		tyP0927LifterMagConv2.tyFB.tyBtnClamp.bValue					:= FALSE;
		tyP0927LifterMagConv2.tyFB.tyBtnUnclamp.bValue				:= FALSE;
	END_IF

	//Mask

	IF p_eLifterMagConv2Status = Error THEN
		fUIInRtStatOff(ADR(tyP0927LifterMagConv2.tyDC.tyBtnMagIn.uiMaskRtStat));
		fUIInRtStatOff(ADR(tyP0927LifterMagConv2.tyDC.tyBtnMagOut.uiMaskRtStat));
		fUIInRtStatOff(ADR(tyP0927LifterMagConv2.tyDC.tyBtnClamp.uiMaskRtStat));
		fUIInRtStatOff(ADR(tyP0927LifterMagConv2.tyDC.tyBtnUnclamp.uiMaskRtStat));

	ELSIF tyP0927LifterMagConv2.tyDC.tyBtnMagIn.bRtCompl = TRUE THEN
		fUIInRtStatHide(ADR(tyP0927LifterMagConv2.tyDC.tyBtnMagIn.uiMaskRtStat));
		fUIInRtStatOff(ADR(tyP0927LifterMagConv2.tyDC.tyBtnMagOut.uiMaskRtStat));
		fUIInRtStatOff(ADR(tyP0927LifterMagConv2.tyDC.tyBtnClamp.uiMaskRtStat));
		fUIInRtStatOff(ADR(tyP0927LifterMagConv2.tyDC.tyBtnUnclamp.uiMaskRtStat));

	ELSIF tyP0927LifterMagConv2.tyDC.tyBtnMagOut.bRtCompl = TRUE THEN
		fUIInRtStatOff(ADR(tyP0927LifterMagConv2.tyDC.tyBtnMagIn.uiMaskRtStat));
		fUIInRtStatHide(ADR(tyP0927LifterMagConv2.tyDC.tyBtnMagOut.uiMaskRtStat));
		fUIInRtStatOff(ADR(tyP0927LifterMagConv2.tyDC.tyBtnClamp.uiMaskRtStat));
		fUIInRtStatOff(ADR(tyP0927LifterMagConv2.tyDC.tyBtnUnclamp.uiMaskRtStat));

	ELSIF tyP0927LifterMagConv2.tyDC.tyBtnStop.bRtCompl = TRUE THEN
		fUIInRtStatHide(ADR(tyP0927LifterMagConv2.tyDC.tyBtnMagIn.uiMaskRtStat));
		fUIInRtStatHide(ADR(tyP0927LifterMagConv2.tyDC.tyBtnMagOut.uiMaskRtStat));
		fUIInRtStatHide(ADR(tyP0927LifterMagConv2.tyDC.tyBtnClamp.uiMaskRtStat));
		fUIInRtStatHide(ADR(tyP0927LifterMagConv2.tyDC.tyBtnUnclamp.uiMaskRtStat));

	END_IF

END_ACTION
```

#### Act_OptP0927RstMnl.st
```iecst
ACTION Act_OptP0927RstMnl:

	IF EDGEPOS((bManualMod = FALSE) OR (p_eLifterMagConv2Status = Error)) THEN

		eLifterMagConv2Act	:= MagConvActIdle;

		//Lifter Mag Conveyor
		//FB
		tyP0927LifterMagConv2.tyFB.tyBtnEnter.bRtCompl				:= FALSE;
		tyP0927LifterMagConv2.tyFB.tyBtnExit.bRtCompl				:= FALSE;
		tyP0927LifterMagConv2.tyFB.tyBtnStop.bRtCompl				:= FALSE;

		tyP0927LifterMagConv2.tyFB.tyBtnEnter.bValue					:= FALSE;
		tyP0927LifterMagConv2.tyFB.tyBtnExit.bValue					:= FALSE;
		tyP0927LifterMagConv2.tyFB.tyBtnStop.bValue					:= TRUE;

		tyP0927LifterMagConv2.tyFB.tyBtnEnter.bRtLk					:= FALSE;
		tyP0927LifterMagConv2.tyFB.tyBtnExit.bRtLk					:= FALSE;
		tyP0927LifterMagConv2.tyFB.tyBtnStop.bRtLk					:= TRUE;

		tyP0927LifterMagConv2.tyFB.tyBtnEnter.uiMaskRtStat.0			:= TRUE;
		tyP0927LifterMagConv2.tyFB.tyBtnExit.uiMaskRtStat.0			:= TRUE;
		tyP0927LifterMagConv2.tyCom.tyBtnDCCtrl.uiMaskRtStat.0		:= TRUE;

		//Direct
		tyP0927LifterMagConv2.tyDC.tyBtnMagIn.bRtCompl				:= FALSE;
		tyP0927LifterMagConv2.tyDC.tyBtnMagOut.bRtCompl				:= FALSE;
		tyP0927LifterMagConv2.tyDC.tyBtnStop.bRtCompl				:= FALSE;

		tyP0927LifterMagConv2.tyDC.tyBtnMagIn.bValue					:= FALSE;
		tyP0927LifterMagConv2.tyDC.tyBtnMagOut.bValue				:= FALSE;
		tyP0927LifterMagConv2.tyDC.tyBtnStop.bValue					:= TRUE;

		tyP0927LifterMagConv2.tyDC.tyBtnMagIn.bRtLk					:= FALSE;
		tyP0927LifterMagConv2.tyDC.tyBtnMagOut.bRtLk					:= FALSE;
		tyP0927LifterMagConv2.tyDC.tyBtnStop.bRtLk					:= TRUE;

		tyP0927LifterMagConv2.tyDC.tyBtnMagIn.uiMaskRtStat.0			:= TRUE;
		tyP0927LifterMagConv2.tyDC.tyBtnMagOut.uiMaskRtStat.0		:= TRUE;
		tyP0927LifterMagConv2.tyCom.tyBtnDCCtrl.uiMaskRtStat.0		:= TRUE;

		//Mag Clamper
		//FB
		tyP0927LifterMagConv2.tyFB.tyBtnClamp.bRtCompl				:= FALSE;
		tyP0927LifterMagConv2.tyFB.tyBtnUnclamp.bRtCompl				:= FALSE;

		tyP0927LifterMagConv2.tyFB.tyBtnClamp.bValue					:= FALSE;
		tyP0927LifterMagConv2.tyFB.tyBtnUnclamp.bValue				:= FALSE;

		tyP0927LifterMagConv2.tyFB.tyBtnClamp.uiMaskRtStat.0			:= TRUE;
		tyP0927LifterMagConv2.tyFB.tyBtnUnclamp.uiMaskRtStat.0		:= TRUE;
		tyP0927LifterMagConv2.tyCom.tyBtnDCCtrl.uiMaskRtStat.0		:= TRUE;

		//Direct
		tyP0927LifterMagConv2.tyDC.tyBtnClamp.bRtCompl				:= FALSE;
		tyP0927LifterMagConv2.tyDC.tyBtnUnclamp.bRtCompl				:= FALSE;

		tyP0927LifterMagConv2.tyDC.tyBtnClamp.bValue					:= FALSE;
		tyP0927LifterMagConv2.tyDC.tyBtnUnclamp.bValue				:= FALSE;

		tyP0927LifterMagConv2.tyDC.tyBtnClamp.uiMaskRtStat.0			:= TRUE;
		tyP0927LifterMagConv2.tyDC.tyBtnUnclamp.uiMaskRtStat.0		:= TRUE;
		tyP0927LifterMagConv2.tyCom.tyBtnDCCtrl.uiMaskRtStat.0		:= TRUE;

	END_IF

	IF EDGEPOS(bManualMod = FALSE) THEN

		tyP0927LifterMagConv2.tyCom.tyBtnDCCtrl.bValue	:= FALSE;

		fUIInRtStatOff(ADR(tyP0927LifterMagConv2.tyFB.tyLyr.uiRtStat));
		fUIInRtStatHide(ADR(tyP0927LifterMagConv2.tyDC.tyLyr.uiRtStat));

	END_IF

END_ACTION
```

#### Act_EntP0928Disp.st
```iecst
ACTION Act_EntP0928Disp:

	//Access Address
	p_tyC0002FullMask ACCESS ADR(tyP0928MagConv.tyFullMaskHide);

	//p_tyC0004Navi ACCESS ADR(tyP0928MagConv.tyNaviBack);

	p_tyC0004Navi ACCESS ADR(tyP0928MagConv.tyNavi2Lyr);

	p_tyC0005Main ACCESS ADR(tyCommon.tyMain);

	p_tyC0007Notif ACCESS ADR(tyCommon.tyNotif);

	p_tyC0008MsgBox ACCESS ADR(tyP0928MagConv.tyMsgBoxHide);

	p_tyC0009Info ACCESS ADR(tyCommon.tyInfo);

	p_tyP0928MagConvCom ACCESS ADR(tyP0928MagConv.tyCom);
	p_tyP0928MagConvTopDC ACCESS ADR(tyP0928MagConv.tyTopDC);
	p_tyP0928MagConvTopFB ACCESS ADR(tyP0928MagConv.tyTopFB);
	p_tyP0928MagConvBtmDC ACCESS ADR(tyP0928MagConv.tyBtmDC);
	p_tyP0928MagConvBtmFB ACCESS ADR(tyP0928MagConv.tyBtmFB);

	IF tyP0928MagConv.tyCom.tyBtnSwitch.bValue AND tyP0928MagConv.tyTopFB.tyLyr.uiRtStat = FALSE THEN
		fUIInRtStatHide(ADR(tyP0928MagConv.tyTopFB.tyLyr.uiRtStat));
		fUIInRtStatOff(ADR(tyP0928MagConv.tyTopDC.tyLyr.uiRtStat));
		fUIInRtStatHide(ADR(tyP0928MagConv.tyBtmFB.tyLyr.uiRtStat));
		fUIInRtStatHide(ADR(tyP0928MagConv.tyBtmDC.tyLyr.uiRtStat));

	ELSIF tyP0928MagConv.tyCom.tyBtnSwitch.bValue AND tyP0928MagConv.tyBtmFB.tyLyr.uiRtStat = FALSE THEN

		fUIInRtStatHide(ADR(tyP0928MagConv.tyTopFB.tyLyr.uiRtStat));
		fUIInRtStatHide(ADR(tyP0928MagConv.tyTopDC.tyLyr.uiRtStat));
		fUIInRtStatHide(ADR(tyP0928MagConv.tyBtmFB.tyLyr.uiRtStat));
		fUIInRtStatOff(ADR(tyP0928MagConv.tyBtmDC.tyLyr.uiRtStat));

	ELSIF tyP0928MagConv.tyCom.tyBtnSwitch.bValue = FALSE AND tyP0928MagConv.tyTopDC.tyLyr.uiRtStat = FALSE THEN
		fUIInRtStatOff(ADR(tyP0928MagConv.tyTopFB.tyLyr.uiRtStat));
		fUIInRtStatHide(ADR(tyP0928MagConv.tyTopDC.tyLyr.uiRtStat));
		fUIInRtStatHide(ADR(tyP0928MagConv.tyBtmFB.tyLyr.uiRtStat));
		fUIInRtStatHide(ADR(tyP0928MagConv.tyBtmDC.tyLyr.uiRtStat));

	ELSIF tyP0928MagConv.tyCom.tyBtnSwitch.bValue = FALSE AND tyP0928MagConv.tyBtmDC.tyLyr.uiRtStat = FALSE THEN
		fUIInRtStatHide(ADR(tyP0928MagConv.tyTopFB.tyLyr.uiRtStat));
		fUIInRtStatHide(ADR(tyP0928MagConv.tyTopDC.tyLyr.uiRtStat));
		fUIInRtStatOff(ADR(tyP0928MagConv.tyBtmFB.tyLyr.uiRtStat));
		fUIInRtStatHide(ADR(tyP0928MagConv.tyBtmDC.tyLyr.uiRtStat));

	END_IF

END_ACTION
```

#### Act_OptP0928FullMask.st
```iecst
ACTION Act_OptP0928FullMask:

	IF eCurrPage = UIP0928MagConv THEN

		IF p_tyDI.bEStopSig = FALSE THEN
			p_tyC0002FullMask ACCESS ADR(tyP0928MagConv.tyFullMaskEStop);

		ELSIF p_tyDI.bCoverSWSig = FALSE THEN
			p_tyC0002FullMask ACCESS ADR(tyP0928MagConv.tyFullMaskCWSig);

		ELSIF p_tyDI.bSafetyRlySig = FALSE THEN
			p_tyC0002FullMask ACCESS ADR(tyP0928MagConv.tyFullMaskSafetyRly);

		ELSE
			p_tyC0002FullMask ACCESS ADR(tyP0928MagConv.tyFullMaskHide);

		END_IF

	END_IF

END_ACTION
```

#### Act_OptP0928Navi.st
```iecst
ACTION Act_OptP0928Navi:

	IF tyP0928MagConv.tyNavi2Lyr.tyBtnBack.bRtCompl = TRUE THEN
		tyP0928MagConv.tyNavi2Lyr.tyBtnBack.bRtCompl	:= FALSE;
		tyP0928MagConv.tyNavi2Lyr.tyBtnBack.bValue		:= FALSE;

		eChgPage	:= UIP0920MtrNPneuCtrl;
	END_IF

	IF p_tyNtParamCurr.bProjMagConvLane1Prep THEN

		IF (tyP0928MagConv.tyNavi2Lyr.tyBtnLeft.bRtCompl OR tyP0928MagConv.tyNavi2Lyr.tyBtnRgt.bRtCompl)
			AND tyP0928MagConv.tyNavi2Lyr.tyBitmapPageDisp.usiValueIdx = 1 THEN
			tyP0928MagConv.tyNavi2Lyr.tyBitmapPageDisp.usiValueIdx := 2;

			tyP0928MagConv.tyNavi2Lyr.tyBtnLeft.bRtCompl	:= FALSE;
			tyP0928MagConv.tyNavi2Lyr.tyBtnLeft.bValue		:= FALSE;
			tyP0928MagConv.tyNavi2Lyr.tyBtnRgt.bRtCompl		:= FALSE;
			tyP0928MagConv.tyNavi2Lyr.tyBtnRgt.bValue		:= FALSE;
			IF tyP0928MagConv.tyCom.tyBtnSwitch.bValue = FALSE THEN
				//Layer (Bottom)
				tyP0928MagConv.tyTopFB.tyLyr.uiRtStat 	:= TRUE;
				tyP0928MagConv.tyTopDC.tyLyr.uiRtStat	:= TRUE;

				tyP0928MagConv.tyBtmFB.tyLyr.uiRtStat 	:= FALSE;
				tyP0928MagConv.tyBtmDC.tyLyr.uiRtStat	:= TRUE;
			ELSE // direct ctrl
				tyP0928MagConv.tyTopFB.tyLyr.uiRtStat 	:= TRUE;
				tyP0928MagConv.tyTopDC.tyLyr.uiRtStat	:= TRUE;

				tyP0928MagConv.tyBtmFB.tyLyr.uiRtStat 	:= TRUE;
				tyP0928MagConv.tyBtmDC.tyLyr.uiRtStat	:= FALSE;
			END_IF
		ELSIF (tyP0928MagConv.tyNavi2Lyr.tyBtnLeft.bRtCompl OR tyP0928MagConv.tyNavi2Lyr.tyBtnRgt.bRtCompl)
			AND tyP0928MagConv.tyNavi2Lyr.tyBitmapPageDisp.usiValueIdx = 2 THEN
			tyP0928MagConv.tyNavi2Lyr.tyBitmapPageDisp.usiValueIdx := 1;

			tyP0928MagConv.tyNavi2Lyr.tyBtnLeft.bRtCompl	:= FALSE;
			tyP0928MagConv.tyNavi2Lyr.tyBtnLeft.bValue		:= FALSE;
			tyP0928MagConv.tyNavi2Lyr.tyBtnRgt.bRtCompl		:= FALSE;
			tyP0928MagConv.tyNavi2Lyr.tyBtnRgt.bValue		:= FALSE;
			IF tyP0928MagConv.tyCom.tyBtnSwitch.bValue = FALSE THEN
				//Layer (Top)
				tyP0928MagConv.tyTopFB.tyLyr.uiRtStat 	:= FALSE;
				tyP0928MagConv.tyTopDC.tyLyr.uiRtStat	:= TRUE;

				tyP0928MagConv.tyBtmFB.tyLyr.uiRtStat 	:= TRUE;
				tyP0928MagConv.tyBtmDC.tyLyr.uiRtStat	:= TRUE;
			ELSE //direct ctrl
				tyP0928MagConv.tyTopFB.tyLyr.uiRtStat 	:= TRUE;
				tyP0928MagConv.tyTopDC.tyLyr.uiRtStat	:= FALSE;

				tyP0928MagConv.tyBtmFB.tyLyr.uiRtStat 	:= TRUE;
				tyP0928MagConv.tyBtmDC.tyLyr.uiRtStat	:= TRUE;
			END_IF
		END_IF

	END_IF
	tyP0928MagConv.tyCom.tyBtnLane.uiRtStat := NOT(p_tyNtParamCurr.bProjMagConvLane2Prep);

	IF tyP0928MagConv.tyCom.tyBtnLane.bRtCompl THEN
		tyP0928MagConv.tyCom.tyBtnLane.bRtCompl := FALSE;
		tyP0928MagConv.tyCom.tyBtnLane.bValue := FALSE;
		eChgPage			:= UIP0929MagConv2;
	END_IF

END_ACTION
```

#### Act_OptP0928MagConv1ChgLyr.st
```iecst
ACTION Act_OptP0928MagConv1ChgLyr:

	IF tyP0928MagConv.tyNavi2Lyr.tyBitmapPageDisp.usiValueIdx = 1 THEN //Top layer

		IF tyP0928MagConv.tyCom.tyBtnSwitch.bRtCompl THEN
			tyP0928MagConv.tyCom.tyBtnSwitch.bRtCompl	:= FALSE;

			IF tyP0928MagConv.tyCom.tyBtnSwitch.bValue = TRUE THEN
				fUIInRtStatOff(ADR(tyP0928MagConv.tyTopDC.tyLyr.uiRtStat));
				fUIInRtStatHide(ADR(tyP0928MagConv.tyTopFB.tyLyr.uiRtStat));
			ELSE
				fUIInRtStatHide(ADR(tyP0928MagConv.tyTopDC.tyLyr.uiRtStat));
				fUIInRtStatOff(ADR(tyP0928MagConv.tyTopFB.tyLyr.uiRtStat));
			END_IF

		END_IF
	ELSIF tyP0928MagConv.tyNavi2Lyr.tyBitmapPageDisp.usiValueIdx = 2 THEN ///Btm layer
		IF tyP0928MagConv.tyCom.tyBtnSwitch.bRtCompl THEN
			tyP0928MagConv.tyCom.tyBtnSwitch.bRtCompl	:= FALSE;

			IF tyP0928MagConv.tyCom.tyBtnSwitch.bValue = TRUE THEN
				fUIInRtStatOff(ADR(tyP0928MagConv.tyBtmDC.tyLyr.uiRtStat));
				fUIInRtStatHide(ADR(tyP0928MagConv.tyBtmFB.tyLyr.uiRtStat));
			ELSE
				fUIInRtStatHide(ADR(tyP0928MagConv.tyBtmDC.tyLyr.uiRtStat));
				fUIInRtStatOff(ADR(tyP0928MagConv.tyBtmFB.tyLyr.uiRtStat));
			END_IF

		END_IF
	END_IF

END_ACTION
```

#### Act_OptP0928MagConv1Sen.st
```iecst
ACTION Act_OptP0928MagConv1Sen:
	// connect sensors to inputs
	tyP0928MagConv.tyCom.tyBtnTopEntSen.bValue			:= p_tyDI.bInMagConvEntSen;
	tyP0928MagConv.tyCom.tyBtnTopMidSen.bValue			:= p_tyDI.bInMagConvMidSen;
	tyP0928MagConv.tyCom.tyBtnTopExtSen.bValue			:= p_tyDI.bInMagConvExtSen;
	tyP0928MagConv.tyCom.tyBtnBtmEntSen.bValue			:= p_tyDI.bOutMagConvEntSen;
	tyP0928MagConv.tyCom.tyBtnBtmMidSen.bValue			:= p_tyDI.bOutMagConvMidSen;
	tyP0928MagConv.tyCom.tyBtnBtmExtSen.bValue			:= p_tyDI.bOutMagConvExtSen;

	//Machine Bitmap
	IF p_tyNtParamCurr.bProjMagConvLane1Prep THEN
		IF tyP0928MagConv.tyNavi2Lyr.tyBitmapPageDisp.usiValueIdx = 1 THEN //Top layer
			tyP0928MagConv.tyCom.tyBitmapMc.uiValueIdx := 0;
		ELSIF tyP0928MagConv.tyNavi2Lyr.tyBitmapPageDisp.usiValueIdx = 2 THEN
			tyP0928MagConv.tyCom.tyBitmapMc.uiValueIdx := 1;
		END_IF
	END_IF

END_ACTION
```

#### Act_OptP0928MagConv1TopFB.st
```iecst
ACTION Act_OptP0928MagConv1TopFB:

	//Magazine Conveyor
	IF tyP0928MagConv.tyTopFB.tyBtnStop.bRtCompl = TRUE THEN
		eInMagConvAct	:= MagConvActStop;

		IF p_eInMagConvStat = MagConvActStop AND p_eInMagConvStatus = Done THEN
			eInMagConvAct	:= MagConvActIdle;

			tyP0928MagConv.tyTopFB.tyBtnEnt.bRtCompl	:= FALSE;
			tyP0928MagConv.tyTopFB.tyBtnEnt.bValue		:= FALSE;
			tyP0928MagConv.tyTopFB.tyBtnEnt.bRtLk		:= FALSE;

			tyP0928MagConv.tyTopFB.tyBtnExit.bRtCompl	:= FALSE;
			tyP0928MagConv.tyTopFB.tyBtnExit.bValue		:= FALSE;
			tyP0928MagConv.tyTopFB.tyBtnExit.bRtLk		:= FALSE;

			tyP0928MagConv.tyTopFB.tyBtnStop.bRtCompl	:= FALSE;
			tyP0928MagConv.tyTopFB.tyBtnStop.bValue		:= TRUE;
			tyP0928MagConv.tyTopFB.tyBtnStop.bRtLk		:= TRUE;
		END_IF

	ELSIF tyP0928MagConv.tyTopFB.tyBtnEnt.bRtCompl = TRUE THEN
		tyP0928MagConv.tyTopFB.tyBtnEnt.bValue	:= TRUE;
		tyP0928MagConv.tyTopFB.tyBtnEnt.bRtLk		:= TRUE;

		tyP0928MagConv.tyTopFB.tyBtnStop.bValue	:= FALSE;
		tyP0928MagConv.tyTopFB.tyBtnStop.bRtLk	:= FALSE;

		eInMagConvAct	:= MagConvActEnt;

		IF p_eInMagConvStat = MagConvActEnt AND p_eInMagConvStatus = Done THEN
			eInMagConvAct	:= MagConvActIdle;

			tyP0928MagConv.tyTopFB.tyBtnEnt.bRtCompl	:= FALSE;

			tyP0928MagConv.tyTopFB.tyBtnEnt.bValue	:= FALSE;
			tyP0928MagConv.tyTopFB.tyBtnEnt.bRtLk		:= FALSE;

			tyP0928MagConv.tyTopFB.tyBtnStop.bValue	:= TRUE;
			tyP0928MagConv.tyTopFB.tyBtnStop.bRtLk	:= TRUE;
		END_IF

	ELSIF tyP0928MagConv.tyTopFB.tyBtnExit.bRtCompl = TRUE THEN
		tyP0928MagConv.tyTopFB.tyBtnExit.bValue	:= TRUE;
		tyP0928MagConv.tyTopFB.tyBtnExit.bRtLk	:= TRUE;

		tyP0928MagConv.tyTopFB.tyBtnStop.bValue	:= FALSE;
		tyP0928MagConv.tyTopFB.tyBtnStop.bRtLk	:= FALSE;

		eInMagConvAct	:= MagConvActExit;

		IF p_eInMagConvStat = MagConvActExit AND p_eInMagConvStatus = Done THEN
			eInMagConvAct	:= MagConvActIdle;

			tyP0928MagConv.tyTopFB.tyBtnExit.bRtCompl:= FALSE;

			tyP0928MagConv.tyTopFB.tyBtnExit.bValue	:= FALSE;
			tyP0928MagConv.tyTopFB.tyBtnExit.bRtLk	:= FALSE;

			tyP0928MagConv.tyTopFB.tyBtnStop.bValue	:= TRUE;
			tyP0928MagConv.tyTopFB.tyBtnStop.bRtLk	:= TRUE;
		END_IF
	END_IF

	//Stopper
	IF tyP0928MagConv.tyCom.tyBtnSwitch.bValue = FALSE THEN

		//Ent Stopper
		IF tyP0928MagConv.tyTopFB.tyBtnEntStprExt.bRtCompl = TRUE THEN
			tyP0928MagConv.tyTopFB.tyBtnEntStprExt.bRtCompl	:= FALSE;

			tyP0928MagConv.tyTopFB.tyBtnEntStprExt.bValue	:= TRUE;
			tyP0928MagConv.tyTopFB.tyBtnEntStprRet.bValue		:= FALSE;

		ELSIF tyP0928MagConv.tyTopFB.tyBtnEntStprRet.bRtCompl = TRUE THEN
			tyP0928MagConv.tyTopFB.tyBtnEntStprRet.bRtCompl	:= FALSE;

			tyP0928MagConv.tyTopFB.tyBtnEntStprRet.bValue		:= TRUE;
			tyP0928MagConv.tyTopFB.tyBtnEntStprExt.bValue	:= FALSE;

		END_IF

		//Mid stopper
		IF tyP0928MagConv.tyTopFB.tyBtnMidStprExt.bRtCompl = TRUE THEN
			tyP0928MagConv.tyTopFB.tyBtnMidStprExt.bRtCompl	:= FALSE;

			tyP0928MagConv.tyTopFB.tyBtnMidStprExt.bValue	:= TRUE;
			tyP0928MagConv.tyTopFB.tyBtnMidStprRet.bValue	:= FALSE;

		ELSIF tyP0928MagConv.tyTopFB.tyBtnMidStprRet.bRtCompl = TRUE THEN
			tyP0928MagConv.tyTopFB.tyBtnMidStprRet.bRtCompl	:= FALSE;

			tyP0928MagConv.tyTopFB.tyBtnMidStprRet.bValue	:= TRUE;
			tyP0928MagConv.tyTopFB.tyBtnMidStprExt.bValue	:= FALSE;

		END_IF

		//Ext Stopper
		IF tyP0928MagConv.tyTopFB.tyBtnExtStprExt.bRtCompl = TRUE THEN
			tyP0928MagConv.tyTopFB.tyBtnExtStprExt.bRtCompl	:= FALSE;

			tyP0928MagConv.tyTopFB.tyBtnExtStprExt.bValue	:= TRUE;
			tyP0928MagConv.tyTopFB.tyBtnExtStprRet.bValue	:= FALSE;

		ELSIF tyP0928MagConv.tyTopFB.tyBtnExtStprRet.bRtCompl = TRUE THEN
			tyP0928MagConv.tyTopFB.tyBtnExtStprRet.bRtCompl	:= FALSE;

			tyP0928MagConv.tyTopFB.tyBtnExtStprRet.bValue	:= TRUE;
			tyP0928MagConv.tyTopFB.tyBtnExtStprExt.bValue	:= FALSE;

		END_IF

		//Action------------
		IF tyP0928MagConv.tyTopFB.tyBtnEntStprExt.bValue = TRUE THEN
			eStopper1Act	:= PneuActExt;

			IF p_eStopper1Stat = PneuActExt AND p_eStopper1Status = Done THEN
				eStopper1Act	:= PneuActIdle;
				tyP0928MagConv.tyTopFB.tyBtnEntStprExt.bValue	:= FALSE;
			ELSIF p_eStopper1Status = Error THEN
				tyP0928MagConv.tyTopFB.tyBtnEntStprExt.bValue	:= FALSE;
			END_IF

		ELSIF tyP0928MagConv.tyTopFB.tyBtnEntStprRet.bValue = TRUE THEN
			eStopper1Act	:= PneuActRet;

			IF p_eStopper1Stat = PneuActRet AND p_eStopper1Status = Done THEN
				eStopper1Act	:= PneuActIdle;
				tyP0928MagConv.tyTopFB.tyBtnEntStprRet.bValue := FALSE;
			ELSIF p_eStopper1Status = Error THEN
				tyP0928MagConv.tyTopFB.tyBtnEntStprRet.bValue := FALSE;
			END_IF

		END_IF

		IF tyP0928MagConv.tyTopFB.tyBtnMidStprExt.bValue = TRUE THEN
			eStopper2Act	:= PneuActExt;

			IF p_eStopper2Stat = PneuActExt AND p_eStopper2Status = Done THEN
				eStopper2Act	:= PneuActIdle;
				tyP0928MagConv.tyTopFB.tyBtnMidStprExt.bValue	:= FALSE;
			ELSIF p_eStopper2Status = Error THEN
				tyP0928MagConv.tyTopFB.tyBtnMidStprExt.bValue	:= FALSE;
			END_IF

		ELSIF tyP0928MagConv.tyTopFB.tyBtnMidStprRet.bValue = TRUE THEN
			eStopper2Act	:= PneuActRet;

			IF p_eStopper2Stat = PneuActRet AND p_eStopper2Status = Done THEN
				eStopper2Act	:= PneuActIdle;
				tyP0928MagConv.tyTopFB.tyBtnMidStprRet.bValue := FALSE;
			ELSIF p_eStopper2Status = Error THEN
				tyP0928MagConv.tyTopFB.tyBtnMidStprRet.bValue := FALSE;
			END_IF

		END_IF

		IF tyP0928MagConv.tyTopFB.tyBtnExtStprExt.bValue = TRUE THEN
			eStopper3Act	:= PneuActExt;

			IF p_eStopper3Stat = PneuActExt AND p_eStopper3Status = Done THEN
				eStopper3Act	:= PneuActIdle;
				tyP0928MagConv.tyTopFB.tyBtnExtStprExt.bValue	:= FALSE;
			ELSIF p_eStopper3Status = Error THEN
				tyP0928MagConv.tyTopFB.tyBtnExtStprExt.bValue	:= FALSE;
			END_IF

		ELSIF tyP0928MagConv.tyTopFB.tyBtnExtStprRet.bValue = TRUE THEN
			eStopper3Act	:= PneuActRet;

			IF p_eStopper3Stat = PneuActRet AND p_eStopper3Status = Done THEN
				eStopper3Act	:= PneuActIdle;
				tyP0928MagConv.tyTopFB.tyBtnExtStprRet.bValue := FALSE;
			ELSIF p_eStopper3Status = Error THEN
				tyP0928MagConv.tyTopFB.tyBtnExtStprRet.bValue := FALSE;
			END_IF

		END_IF

		//Update Status
//		tyP0928MagConv.tyDC.tyBtnFixedUnclamp.bValue	:= NOT p_bStopper1RetCtrl2;
//		tyP0928MagConv.tyDC.tyBtnFixedClamp.bValue		:= p_bMagConv2Clp1ClprFixClampCtrl;
//		tyP0928MagConv.tyDC.tyBtnRemoteUnclamp.bValue	:= NOT p_bMagConv2Clp1ClprRmtClampCtrl;
//		tyP0928MagConv.tyDC.tyBtnRemoteClamp.bValue	:= p_bMagConv2Clp1ClprRmtClampCtrl;
//
//		tyP0928MagConv.tyDC.tyBtnSelUnclamp.bRtCompl	:= FALSE;
//		tyP0928MagConv.tyDC.tyBtnSelClamp.bRtCompl		:= FALSE;
//		tyP0928MagConv.tyDC.tyBtnSelUnclamp.bValue	:= p_bSelClamp1RetCtrl;
//		tyP0928MagConv.tyDC.tyBtnSelClamp.bValue	:= p_bSelClamp1ExtCtrl;
	END_IF

	//Mask
//	IF p_tyUsrMgmtCurrAccessRgt.bManualFBOnly THEN
//
//		fUIInRtStatOff(ADR(tyP0928MagConv.tyCom.tyBtnSwitch.uiMaskRtStat));
//
//	ELSE
//
//		IF p_eInMagConvStatus = Error THEN
//
//			fUIInRtStatOff(ADR(tyP0928MagConv.tyTopFB.tyBtnEnt.uiMaskRtStat));
//			fUIInRtStatOff(ADR(tyP0928MagConv.tyTopFB.tyBtnExit.uiMaskRtStat));
//			fUIInRtStatOff(ADR(tyP0928MagConv.tyTopFB.tyBtnEntStprExt.uiMaskRtStat));
//			fUIInRtStatOff(ADR(tyP0928MagConv.tyTopFB.tyBtnEntStprRet.uiMaskRtStat));
//			fUIInRtStatOff(ADR(tyP0928MagConv.tyTopFB.tyBtnMidStprExt.uiMaskRtStat));
//			fUIInRtStatOff(ADR(tyP0928MagConv.tyTopFB.tyBtnMidStprRet.uiMaskRtStat));
//			fUIInRtStatOff(ADR(tyP0928MagConv.tyTopFB.tyBtnExtStprExt.uiMaskRtStat));
//			fUIInRtStatOff(ADR(tyP0928MagConv.tyTopFB.tyBtnExtStprRet.uiMaskRtStat));
//			fUIInRtStatHide(ADR(tyP0928MagConv.tyCom.tyBtnSwitch.uiMaskRtStat));
//
//		ELSIF tyP0928MagConv.tyTopFB.tyBtnEnt.bRtCompl = TRUE THEN
//
//			fUIInRtStatHide(ADR(tyP0928MagConv.tyTopFB.tyBtnEnt.uiMaskRtStat));
//			fUIInRtStatOff(ADR(tyP0928MagConv.tyTopFB.tyBtnExit.uiMaskRtStat));
//			fUIInRtStatOff(ADR(tyP0928MagConv.tyTopFB.tyBtnFixedClamp.uiMaskRtStat));
//			fUIInRtStatOff(ADR(tyP0928MagConv.tyTopFB.tyBtnFixedUnclamp.uiMaskRtStat));
//			fUIInRtStatOff(ADR(tyP0928MagConv.tyTopFB.tyBtnRemoteClamp.uiMaskRtStat));
//			fUIInRtStatOff(ADR(tyP0928MagConv.tyTopFB.tyBtnRemoteUnclamp.uiMaskRtStat));
//			fUIInRtStatOff(ADR(tyP0928MagConv.tyTopFB.tyBtnSelClamp.uiMaskRtStat));
//			fUIInRtStatOff(ADR(tyP0928MagConv.tyTopFB.tyBtnSelUnclamp.uiMaskRtStat));
//			fUIInRtStatOff(ADR(tyP0928MagConv.tyCom.tyBtnSwitch.uiMaskRtStat));
//
//		ELSIF tyP0928MagConv.tyTopFB.tyBtnExit.bRtCompl = TRUE THEN
//
//			fUIInRtStatOff(ADR(tyP0928MagConv.tyTopFB.tyBtnEnt.uiMaskRtStat));
//			fUIInRtStatHide(ADR(tyP0928MagConv.tyTopFB.tyBtnExit.uiMaskRtStat));
//			fUIInRtStatOff(ADR(tyP0928MagConv.tyTopFB.tyBtnFixedClamp.uiMaskRtStat));
//			fUIInRtStatOff(ADR(tyP0928MagConv.tyTopFB.tyBtnFixedUnclamp.uiMaskRtStat));
//			fUIInRtStatOff(ADR(tyP0928MagConv.tyTopFB.tyBtnRemoteClamp.uiMaskRtStat));
//			fUIInRtStatOff(ADR(tyP0928MagConv.tyTopFB.tyBtnRemoteUnclamp.uiMaskRtStat));
//			fUIInRtStatOff(ADR(tyP0928MagConv.tyTopFB.tyBtnSelClamp.uiMaskRtStat));
//			fUIInRtStatOff(ADR(tyP0928MagConv.tyTopFB.tyBtnSelUnclamp.uiMaskRtStat));
//			fUIInRtStatOff(ADR(tyP0928MagConv.tyCom.tyBtnSwitch.uiMaskRtStat));
//
//		ELSIF tyP0928MagConv.tyTopFB.tyBtnFixedClamp.bValue = TRUE OR tyP0928MagConv.tyTopFB.tyBtnRemoteClamp.bValue = TRUE
//			OR tyP0928MagConv.tyTopFB.tyBtnFixedUnclamp.bValue = TRUE OR tyP0928MagConv.tyTopFB.tyBtnRemoteUnclamp.bValue = TRUE
//			OR tyP0928MagConv.tyTopFB.tyBtnSelUnclamp.bValue = TRUE OR tyP0928MagConv.tyTopFB.tyBtnSelClamp.bValue = TRUE
//			THEN
//
//			fUIInRtStatOff(ADR(tyP0928MagConv.tyTopFB.tyBtnEnt.uiMaskRtStat));
//			fUIInRtStatOff(ADR(tyP0928MagConv.tyTopFB.tyBtnExit.uiMaskRtStat));
//			fUIInRtStatHide(ADR(tyP0928MagConv.tyTopFB.tyBtnFixedClamp.uiMaskRtStat));
//		fUIInRtStatHide(ADR(tyP0928MagConv.tyTopFB.tyBtnFixedUnclamp.uiMaskRtStat));
//		fUIInRtStatHide(ADR(tyP0928MagConv.tyTopFB.tyBtnRemoteClamp.uiMaskRtStat));
//		fUIInRtStatHide(ADR(tyP0928MagConv.tyTopFB.tyBtnRemoteUnclamp.uiMaskRtStat));
//		fUIInRtStatHide(ADR(tyP0928MagConv.tyTopFB.tyBtnSelClamp.uiMaskRtStat));
//		fUIInRtStatHide(ADR(tyP0928MagConv.tyTopFB.tyBtnSelUnclamp.uiMaskRtStat));
//		fUIInRtStatOff(ADR(tyP0928MagConv.tyCom.tyBtnSwitch.uiMaskRtStat));
//
//	ELSE
//
//		fUIInRtStatHide(ADR(tyP0928MagConv.tyTopFB.tyBtnEnt.uiMaskRtStat));
//		fUIInRtStatHide(ADR(tyP0928MagConv.tyTopFB.tyBtnExit.uiMaskRtStat));
//		fUIInRtStatHide(ADR(tyP0928MagConv.tyTopFB.tyBtnFixedClamp.uiMaskRtStat));
//		fUIInRtStatHide(ADR(tyP0928MagConv.tyTopFB.tyBtnFixedUnclamp.uiMaskRtStat));
//		fUIInRtStatHide(ADR(tyP0928MagConv.tyTopFB.tyBtnRemoteClamp.uiMaskRtStat));
//		fUIInRtStatHide(ADR(tyP0928MagConv.tyTopFB.tyBtnRemoteUnclamp.uiMaskRtStat));
//		fUIInRtStatHide(ADR(tyP0928MagConv.tyTopFB.tyBtnSelClamp.uiMaskRtStat));
//		fUIInRtStatHide(ADR(tyP0928MagConv.tyTopFB.tyBtnSelUnclamp.uiMaskRtStat));
//		fUIInRtStatHide(ADR(tyP0928MagConv.tyCom.tyBtnSwitch.uiMaskRtStat));
//
//	END_IF
//END_IF

END_ACTION
```

#### Act_OptP0928MagConv1FBStat.st
```iecst
ACTION Act_OptP0928MagConv1FBStat:

	IF tyP0928MagConv.tyTopFB.tyBtnEntStprExt.bValue OR tyP0928MagConv.tyTopFB.tyBtnEntStprRet.bValue THEN
		tyP0928MagConv.tyTopFB.tyStringStat.sValue	:= p_sStopper1StatTxt;
	ELSIF tyP0928MagConv.tyTopFB.tyBtnMidStprExt.bValue OR tyP0928MagConv.tyTopFB.tyBtnMidStprRet.bValue THEN
		tyP0928MagConv.tyTopFB.tyStringStat.sValue	:= p_sStopper2StatTxt;
	ELSIF tyP0928MagConv.tyTopFB.tyBtnExtStprExt.bValue OR tyP0928MagConv.tyTopFB.tyBtnExtStprRet.bValue THEN
		tyP0928MagConv.tyTopFB.tyStringStat.sValue	:= p_sStopper3StatTxt;

	ELSIF tyP0928MagConv.tyBtmFB.tyBtnMidStprExt.bValue OR tyP0928MagConv.tyBtmFB.tyBtnMidStprRet.bValue THEN
		tyP0928MagConv.tyBtmFB.tyStringStat.sValue	:= p_sStopper4StatTxt;
	ELSIF tyP0928MagConv.tyBtmFB.tyBtnExtStprExt.bValue OR tyP0928MagConv.tyBtmFB.tyBtnExtStprRet.bValue THEN
		tyP0928MagConv.tyBtmFB.tyStringStat.sValue	:= p_sStopper5StatTxt;

	ELSIF tyP0928MagConv.tyTopFB.tyBtnEnt.bValue OR tyP0928MagConv.tyTopFB.tyBtnExit.bValue THEN
		tyP0928MagConv.tyTopFB.tyStringStat.sValue	:= p_sInMagConvStatTxt;
	ELSIF tyP0928MagConv.tyBtmFB.tyBtnEnt.bValue OR tyP0928MagConv.tyBtmFB.tyBtnExit.bValue THEN
		tyP0928MagConv.tyBtmFB.tyStringStat.sValue	:= p_sOutMagConvStatTxt;

	END_IF

END_ACTION
```
